FB_AlarmCodeManager(
bAlarm1         :=MesIO_SUBMV_EL1809_1[ 1].value , // SUBMV.-EL1809-ID:1-Input:1 : MV Feeder 1 Opened #Interface
bAlarm2         :=MesIO_SUBMV_EL1809_1[ 2].value , //SUBMV.-EL1809-ID:1-Input:2 : MV Feeder 2 Opened #Interface
bAlarm3         :=MesIO_SUBMV_EL1809_1[ 3].value , //SUBMV.-EL1809-ID:1-Input:3 : MV Feeder 3 Opened  #Interface
bAlarm4         :=MesIO_SUBMV_EL1809_1[ 4].value , //SUBMV.-EL1809-ID:1-Input:4 : Main MVCB Opened #Interface
bAlarm5         :=MesIO_SUBMV_EL1809_1[ 5].value , //SUBMV.-EL1809-ID:1-Input:5 : MainMVCB Tripped #Interface
bAlarm6         :=MesIO_SUBMV_EL1809_1[ 6].value , //SUBMV.-EL1809-ID:1-Input:6 : MainMVCB Earthing #Interface
bAlarm7         :=MesIO_SUBMV_EL1809_1[ 7].value , //SUBMV.-EL1809-ID:1-Input:7 : MainMVCB selector in local position #Interface
bAlarm8         :=MesIO_SUBMV_EL1809_1[ 8].value , //SUBMV.-EL1809-ID:1-Input:8 : MainMVCB motorization in fault #Interface
bAlarm9         :=MesIO_SUBMV_EL1809_1[ 9].value , //SUBMV.-EL1809-ID:1-Input:9 : MV Feeder 1 Tripped #Interface
bAlarm10         :=MesIO_SUBMV_EL1809_1[ 10].value , //SUBMV.-EL1809-ID:1-Input:10 : MV Feeder 2 Tripped #Interface
bAlarm11         :=MesIO_SUBMV_EL1809_1[ 11].value , //SUBMV.-EL1809-ID:1-Input:11 : MV Feeder 3 Tripped  #Interface
bAlarm12         :=MesIO_SUBMV_EL1809_1[ 12].value , //SUBMV.-EL1809-ID:1-Input:12 : MV Feeder 1 Motorization fault #Interface
bAlarm13         :=MesIO_SUBMV_EL1809_1[ 13].value , //SUBMV.-EL1809-ID:1-Input:13 : MV Feeder 2 Motorization fault #Interface
bAlarm14         :=MesIO_SUBMV_EL1809_1[ 14].value , //SUBMV.-EL1809-ID:1-Input:14 : MV Feeder 3 Motorization fault  #Interface
bAlarm15         :=MesIO_SUBMV_EL1809_1[ 15].value , //SUBMV.-EL1809-ID:1-Input:15 : MV Feeder 1 Earthing #Interface
wAlarmCode      => MesData.MesEventCode[1]);   
FB_AlarmCodeManager(
bAlarm1         :=MesIO_SUBMV_EL1809_1[ 16].value , //SUBMV.-EL1809-ID:1-Input:16 : MV Feeder 2 Earthing #Interface
bAlarm2         :=MesIO_SUBMV_EL1809_2[ 1].value , //SUBMV.-EL1809-ID:2-Input:1 : MV Feeder 3 Earthing  #Interface
bAlarm3         :=MesIO_SUBMV_EL1809_2[ 2].value , //SUBMV.-EL1809-ID:2-Input:2 : MV Feeder 1 Selector in local position #Interface
bAlarm4         :=MesIO_SUBMV_EL1809_2[ 3].value , //SUBMV.-EL1809-ID:2-Input:3 : MV Feeder 2 Selector in local position #Interface
bAlarm5         :=MesIO_SUBMV_EL1809_2[ 4].value , //SUBMV.-EL1809-ID:2-Input:4 : MV Feeder 3 Selector in local position  #Interface
bAlarm6         :=MesIO_SUBMV_EL1809_2[ 5].value , //SUBMV.-EL1809-ID:2-Input:5 : Grid MV CB opened #Interface
bAlarm7         :=MesIO_SUBMV_EL1809_2[ 6].value , //SUBMV.-EL1809-ID:2-Input:6 : Measure MV CB opened  #Interface
bAlarm8         :=MesIO_SUBMV_EL1809_2[ 7].value , //SUBMV.-EL1809-ID:2-Input:7 : Measure MV CB Fuse is burned #Interface
bAlarm9         :=MesIO_SUBMV_EL1809_2[ 8].value , //SUBMV.-EL1809-ID:2-Input:8 : Measure MVCB Earthing #Interface
bAlarm10         :=MesIO_SUBMV_EL1809_2[ 9].value , //SUBMV.-EL1809-ID:2-Input:9 : AuxMVCB opened #Interface
bAlarm11         :=MesIO_SUBMV_EL1809_2[ 10].value , //SUBMV.-EL1809-ID:2-Input:10 : AuxMVCB fuse is burned #Interface
bAlarm12         :=MesIO_SUBMV_EL1809_2[ 11].value , //SUBMV.-EL1809-ID:2-Input:11 : AuxMVCB earthing #Interface
bAlarm13         :=MesIO_SUBMV_EL1809_2[ 12].value , //SUBMV.-EL1809-ID:2-Input:12 : Emergency Stop in LV Area #Interface
bAlarm14         :=MesIO_SUBMV_EL1809_2[ 13].value , //SUBMV.-EL1809-ID:2-Input:13 : Emergency stop in MV Area #Interface
bAlarm15         :=MesIO_SUBMV_EL1809_2[ 14].value , //SUBMV.-EL1809-ID:2-Input:14 : Smoke detector in LV Area #Interface
wAlarmCode      => MesData.MesEventCode[2]);   
FB_AlarmCodeManager(
bAlarm1         :=MesIO_SUBMV_EL1809_2[ 16].value , //SUBMV.-EL1809-ID:2-Input:16 : Transformer Alarm synthesis #Interface
bAlarm2         :=MesIO_SUBMV_EL1809_3[ 1].value , //SUBMV.-EL1809-ID:3-Input:1 : Transformer pressure alarm #Interface
bAlarm3         :=MesIO_SUBMV_EL1809_3[ 2].value , //SUBMV.-EL1809-ID:3-Input:2 : Transformer gaz alarm  #Interface
bAlarm4         :=MesIO_SUBMV_EL1809_3[ 3].value , //SUBMV.-EL1809-ID:3-Input:3 : Transformer temperature warning  #Interface
bAlarm5         :=MesIO_SUBMV_EL1809_3[ 4].value , //SUBMV.-EL1809-ID:3-Input:4 : Transformer temperature alarm #Interface
bAlarm6         :=MesIO_SUBMV_EL1809_3[ 5].value , //SUBMV.-EL1809-ID:3-Input:5 : UPS Decharge Batterie State #Interface
bAlarm7         :=MesIO_SUBMV_EL1809_3[ 6].value , //SUBMV.-EL1809-ID:3-Input:6 : UPS alarm synthesis #Interface
bAlarm8         :=MesIO_SUBMV_EL1809_3[ 7].value , //SUBMV.-EL1809-ID:3-Input:7 : UPS  Low Voltage  #Interface
bAlarm9         :=MesIO_SUBMV_EL1809_3[ 8].value , //SUBMV.-EL1809-ID:3-Input:8 : ProtectRelay I>>0 Fault #Interface
bAlarm10         :=MesIO_SUBMV_EL1809_3[ 9].value , //SUBMV.-EL1809-ID:3-Input:9 : ProtectRelay Min U Fault #Interface
bAlarm11         :=MesIO_SUBMV_EL2809_4[ 1].value , //SUBMV.-EL2809-ID:4-Output:1 : MainMVCB Open order #Interface
bAlarm12         :=MesIO_SUBMV_EL2809_4[ 2].value , //SUBMV.-EL2809-ID:4-Output:2 : MainMVCB Close order #Interface
bAlarm13         :=MesIO_SUBMV_EL2809_4[ 3].value , //SUBMV.-EL2809-ID:4-Output:3 : MV Feeder 1 Close Command #Interface
bAlarm14         :=MesIO_SUBMV_EL2809_4[ 4].value , //SUBMV.-EL2809-ID:4-Output:4 : MV Feeder 2 Close Command #Interface
bAlarm15         :=MesIO_SUBMV_EL2809_4[ 5].value , //SUBMV.-EL2809-ID:4-Output:5 : MV Feeder 3 Close Command  #Interface
wAlarmCode      => MesData.MesEventCode[3]);   
FB_AlarmCodeManager(
bAlarm1         :=MesIO_SUBMV_EL2809_4[ 6].value , //SUBMV.-EL2809-ID:4-Output:6 : MV Feeder 1 Open Command #Interface
bAlarm2         :=MesIO_SUBMV_EL2809_4[ 7].value , //SUBMV.-EL2809-ID:4-Output:7 : MV Feeder 2 Open Command #Interface
bAlarm3         :=MesIO_SUBMV_EL2809_4[ 8].value , //SUBMV.-EL2809-ID:4-Output:8 : MV Feeder 3 Open Command  #Interface
bAlarm4         :=MesIO_PTR_1_EL1809_9[ 1].value , //PTR.1-EL1809-ID:9-Input:1 : Motorization alarm MainMVCB #Interface
bAlarm5         :=MesIO_PTR_1_EL1809_9[ 2].value , //PTR.1-EL1809-ID:9-Input:2 : Main MVCB Tripped #Interface
bAlarm6         :=MesIO_PTR_1_EL1809_9[ 3].value , //PTR.1-EL1809-ID:9-Input:3 : MainMVCB selector in Local position #Interface
bAlarm7         :=MesIO_PTR_1_EL1809_9[ 4].value , //PTR.1-EL1809-ID:9-Input:4 : MainMVCB connected to the Earth #Interface
bAlarm8         :=MesIO_PTR_1_EL1809_9[ 5].value , //PTR.1-EL1809-ID:9-Input:5 : Transfo smoke detector 1 #Interface
bAlarm9         :=MesIO_PTR_1_EL1809_9[ 6].value , //PTR.1-EL1809-ID:9-Input:6 : Inverter smoke detector 2 #Interface
bAlarm10         :=MesIO_PTR_1_EL1809_9[ 7].value , //PTR.1-EL1809-ID:9-Input:7 : Door sensor Transformer  area #Interface
bAlarm11         :=MesIO_PTR_1_EL1809_9[ 8].value , //PTR.1-EL1809-ID:9-Input:8 : Door sensor inverter area #Interface
bAlarm12         :=MesIO_PTR_1_EL1809_9[ 9].value , //PTR.1-EL1809-ID:9-Input:9 : Transformer Alarm synthesis #Interface
bAlarm13         :=MesIO_PTR_1_EL1809_9[ 10].value , //PTR.1-EL1809-ID:9-Input:10 : Transformer pressure alarm #Interface
bAlarm14         :=MesIO_PTR_1_EL1809_9[ 11].value , //PTR.1-EL1809-ID:9-Input:11 : Transformer gaz alarm  #Interface
bAlarm15         :=MesIO_PTR_1_EL1809_9[ 12].value , //PTR.1-EL1809-ID:9-Input:12 : Transformer temperature warning  #Interface
wAlarmCode      => MesData.MesEventCode[4]);   
FB_AlarmCodeManager(
bAlarm1         :=MesIO_PTR_1_EL1809_9[ 13].value , //PTR.1-EL1809-ID:9-Input:13 : Transformer temperature alarm #Interface
bAlarm2         :=MesIO_PTR_1_EL1809_9[ 14].value , //PTR.1-EL1809-ID:9-Input:14 : Auxiliairy main CB Opened #Interface
bAlarm3         :=MesIO_PTR_1_EL2809_10[ 1].value , //PTR.1-EL2809-ID:10-Output:1 : Open Command MainMVCB #Interface
bAlarm4         :=MesIO_PTR_1_EL2809_10[ 2].value , //PTR.1-EL2809-ID:10-Output:2 : Close Command MainMVCB #Interface
bAlarm5         :=MesIO_PTR_2_EL1809_9[ 1].value , //PTR.2-EL1809-ID:9-Input:1 : Motorization alarm MainMVCB #Interface
bAlarm6         :=MesIO_PTR_2_EL1809_9[ 2].value , //PTR.2-EL1809-ID:9-Input:2 : Main MVCB Tripped #Interface
bAlarm7         :=MesIO_PTR_2_EL1809_9[ 3].value , //PTR.2-EL1809-ID:9-Input:3 : MainMVCB selector in Local position #Interface
bAlarm8         :=MesIO_PTR_2_EL1809_9[ 4].value , //PTR.2-EL1809-ID:9-Input:4 : MainMVCB connected to the Earth #Interface
bAlarm9         :=MesIO_PTR_2_EL1809_9[ 5].value , //PTR.2-EL1809-ID:9-Input:5 : Transfo smoke detector 1 #Interface
bAlarm10         :=MesIO_PTR_2_EL1809_9[ 6].value , //PTR.2-EL1809-ID:9-Input:6 : Inverter smoke detector 2 #Interface
bAlarm11         :=MesIO_PTR_2_EL1809_9[ 7].value , //PTR.2-EL1809-ID:9-Input:7 : Door sensor Transformer  area #Interface
bAlarm12         :=MesIO_PTR_2_EL1809_9[ 8].value , //PTR.2-EL1809-ID:9-Input:8 : Door sensor inverter area #Interface
bAlarm13         :=MesIO_PTR_2_EL1809_9[ 9].value , //PTR.2-EL1809-ID:9-Input:9 : Transformer Alarm synthesis #Interface
bAlarm14         :=MesIO_PTR_2_EL1809_9[ 10].value , //PTR.2-EL1809-ID:9-Input:10 : Transformer pressure alarm #Interface
bAlarm15         :=MesIO_PTR_2_EL1809_9[ 11].value , //PTR.2-EL1809-ID:9-Input:11 : Transformer gaz alarm  #Interface
wAlarmCode      => MesData.MesEventCode[5]);   
FB_AlarmCodeManager(
bAlarm1         :=MesIO_PTR_2_EL1809_9[ 12].value , //PTR.2-EL1809-ID:9-Input:12 : Transformer temperature warning  #Interface
bAlarm2         :=MesIO_PTR_2_EL1809_9[ 13].value , //PTR.2-EL1809-ID:9-Input:13 : Transformer temperature alarm #Interface
bAlarm3         :=MesIO_PTR_2_EL1809_9[ 14].value , //PTR.2-EL1809-ID:9-Input:14 : Auxiliairy main CB Opened #Interface
bAlarm4         :=MesIO_PTR_2_EL2809_10[ 1].value , //PTR.2-EL2809-ID:10-Output:1 : Open Command MainMVCB #Interface
bAlarm5         :=MesIO_PTR_2_EL2809_10[ 2].value , //PTR.2-EL2809-ID:10-Output:2 : Close Command MainMVCB #Interface
bAlarm6         :=MesIO_PTR_3_EL1809_9[ 1].value , //PTR.3-EL1809-ID:9-Input:1 : Motorization alarm MainMVCB #Interface
bAlarm7         :=MesIO_PTR_3_EL1809_9[ 2].value , //PTR.3-EL1809-ID:9-Input:2 : Main MVCB Tripped #Interface
bAlarm8         :=MesIO_PTR_3_EL1809_9[ 3].value , //PTR.3-EL1809-ID:9-Input:3 : MainMVCB selector in Local position #Interface
bAlarm9         :=MesIO_PTR_3_EL1809_9[ 4].value , //PTR.3-EL1809-ID:9-Input:4 : MainMVCB connected to the Earth #Interface
bAlarm10         :=MesIO_PTR_3_EL1809_9[ 5].value , //PTR.3-EL1809-ID:9-Input:5 : Transfo smoke detector 1 #Interface
bAlarm11         :=MesIO_PTR_3_EL1809_9[ 6].value , //PTR.3-EL1809-ID:9-Input:6 : Inverter smoke detector 2 #Interface
bAlarm12         :=MesIO_PTR_3_EL1809_9[ 7].value , //PTR.3-EL1809-ID:9-Input:7 : Door sensor Transformer  area #Interface
bAlarm13         :=MesIO_PTR_3_EL1809_9[ 8].value , //PTR.3-EL1809-ID:9-Input:8 : Door sensor inverter area #Interface
bAlarm14         :=MesIO_PTR_3_EL1809_9[ 9].value , //PTR.3-EL1809-ID:9-Input:9 : Transformer Alarm synthesis #Interface
bAlarm15         :=MesIO_PTR_3_EL1809_9[ 10].value , //PTR.3-EL1809-ID:9-Input:10 : Transformer pressure alarm #Interface
wAlarmCode      => MesData.MesEventCode[6]);   
FB_AlarmCodeManager(
bAlarm1         :=MesIO_PTR_3_EL1809_9[ 11].value , //PTR.3-EL1809-ID:9-Input:11 : Transformer gaz alarm  #Interface
bAlarm2         :=MesIO_PTR_3_EL1809_9[ 12].value , //PTR.3-EL1809-ID:9-Input:12 : Transformer temperature warning  #Interface
bAlarm3         :=MesIO_PTR_3_EL1809_9[ 13].value , //PTR.3-EL1809-ID:9-Input:13 : Transformer temperature alarm #Interface
bAlarm4         :=MesIO_PTR_3_EL1809_9[ 14].value , //PTR.3-EL1809-ID:9-Input:14 : Auxiliairy main CB Opened #Interface
bAlarm5         :=MesIO_PTR_3_EL2809_10[ 1].value , //PTR.3-EL2809-ID:10-Output:1 : Open Command MainMVCB #Interface
bAlarm6         :=MesIO_PTR_3_EL2809_10[ 2].value , //PTR.3-EL2809-ID:10-Output:2 : Close Command MainMVCB #Interface
wAlarmCode      => MesData.MesEventCode[7]);
END_METHOD

METHOD M_Evaluate : BOOL
(*
MesIO_SUBMV_EL1809_1[1].value := axDI[1] ;
MesIO_SUBMV_EL1809_1[2].value := axDI[2] ;
MesIO_SUBMV_EL1809_1[3].value := axDI[3] ;
MesIO_SUBMV_EL1809_1[4].value := axDI[4] ;
MesIO_SUBMV_EL1809_1[5].value := axDI[5] ;
MesIO_SUBMV_EL1809_1[6].value := axDI[6] ;
MesIO_SUBMV_EL1809_1[7].value := axDI[7] ;
MesIO_SUBMV_EL1809_1[8].value := axDI[8] ;
MesIO_SUBMV_EL1809_1[9].value := axDI[9] ;
MesIO_SUBMV_EL1809_1[10].value := axDI[10] ;
MesIO_SUBMV_EL1809_1[11].value := axDI[11] ;
MesIO_SUBMV_EL1809_1[12].value := axDI[12] ;
MesIO_SUBMV_EL1809_1[13].value := axDI[13] ;
MesIO_SUBMV_EL1809_1[14].value := axDI[14] ;
MesIO_SUBMV_EL1809_1[15].value := axDI[15] ;
MesIO_SUBMV_EL1809_1[16].value := axDI[16] ;
MesIO_SUBMV_EL1809_2[1].value := axDI[17] ;
MesIO_SUBMV_EL1809_2[2].value := axDI[18] ;
MesIO_SUBMV_EL1809_2[3].value := axDI[19] ;
MesIO_SUBMV_EL1809_2[4].value := axDI[20] ;
MesIO_SUBMV_EL1809_2[5].value := axDI[21] ;
MesIO_SUBMV_EL1809_2[6].value := axDI[22] ;
MesIO_SUBMV_EL1809_2[7].value := axDI[23] ;
MesIO_SUBMV_EL1809_2[8].value := axDI[24] ;
MesIO_SUBMV_EL1809_2[9].value := axDI[25] ;
MesIO_SUBMV_EL1809_2[10].value := axDI[26] ;
MesIO_SUBMV_EL1809_2[11].value := axDI[27] ;
MesIO_SUBMV_EL1809_2[12].value := axDI[28] ;
MesIO_SUBMV_EL1809_2[13].value := axDI[29] ;
MesIO_SUBMV_EL1809_2[14].value := axDI[30] ;
MesIO_SUBMV_EL1809_2[15].value := axDI[31] ;
MesIO_SUBMV_EL1809_2[16].value := axDI[32] ;
MesIO_SUBMV_EL1809_3[1].value := axDI[33] ;
MesIO_SUBMV_EL1809_3[2].value := axDI[34] ;
MesIO_SUBMV_EL1809_3[3].value := axDI[35] ;
MesIO_SUBMV_EL1809_3[4].value := axDI[36] ;
MesIO_SUBMV_EL1809_3[5].value := axDI[37] ;
MesIO_SUBMV_EL1809_3[6].value := axDI[38] ;
MesIO_SUBMV_EL1809_3[7].value := axDI[39] ;
MesIO_SUBMV_EL1809_3[8].value := axDI[40] ;
MesIO_SUBMV_EL1809_3[9].value := axDI[41] ;
MesIO_SUBMV_EL1809_3[10].value := axDI[42] ;
MesIO_SUBMV_EL1809_3[11].value := axDI[43] ;
MesIO_SUBMV_EL1809_3[12].value := axDI[44] ;
MesIO_SUBMV_EL1809_3[13].value := axDI[45] ;
MesIO_SUBMV_EL1809_3[14].value := axDI[46] ;
MesIO_SUBMV_EL1809_3[15].value := axDI[47] ;
MesIO_SUBMV_EL1809_3[16].value := axDI[48] ;
axDO[1] := MesIO_SUBMV_EL2809_4[1].value ; 
axDO[2] := MesIO_SUBMV_EL2809_4[2].value ; 
axDO[3] := MesIO_SUBMV_EL2809_4[3].value ; 
axDO[4] := MesIO_SUBMV_EL2809_4[4].value ; 
axDO[5] := MesIO_SUBMV_EL2809_4[5].value ; 
axDO[6] := MesIO_SUBMV_EL2809_4[6].value ; 
axDO[7] := MesIO_SUBMV_EL2809_4[7].value ; 
axDO[8] := MesIO_SUBMV_EL2809_4[8].value ; 
axDO[9] := MesIO_SUBMV_EL2809_4[9].value ; 
axDO[10] := MesIO_SUBMV_EL2809_4[10].value ; 
axDO[11] := MesIO_SUBMV_EL2809_4[11].value ; 
axDO[12] := MesIO_SUBMV_EL2809_4[12].value ; 
axDO[13] := MesIO_SUBMV_EL2809_4[13].value ; 
axDO[14] := MesIO_SUBMV_EL2809_4[14].value ; 
axDO[15] := MesIO_SUBMV_EL2809_4[15].value ; 
axDO[16] := MesIO_SUBMV_EL2809_4[16].value ; 
MesIO_SUBMV_EL3024_5[1].value := axAI[1] ;
MesIO_SUBMV_EL3024_5[2].value := axAI[2] ;
MesIO_SUBMV_EL3024_5[3].value := axAI[3] ;
MesIO_SUBMV_EL3024_5[4].value := axAI[4] ;
MesIO_PTR_1_EL3024_8[1].value := axAI[5] ;
MesIO_PTR_1_EL3024_8[2].value := axAI[6] ;
MesIO_PTR_1_EL3024_8[3].value := axAI[7] ;
MesIO_PTR_1_EL3024_8[4].value := axAI[8] ;
MesIO_PTR_1_EL1809_9[1].value := axDI[49] ;
MesIO_PTR_1_EL1809_9[2].value := axDI[50] ;
MesIO_PTR_1_EL1809_9[3].value := axDI[51] ;
MesIO_PTR_1_EL1809_9[4].value := axDI[52] ;
MesIO_PTR_1_EL1809_9[5].value := axDI[53] ;
MesIO_PTR_1_EL1809_9[6].value := axDI[54] ;
MesIO_PTR_1_EL1809_9[7].value := axDI[55] ;
MesIO_PTR_1_EL1809_9[8].value := axDI[56] ;
MesIO_PTR_1_EL1809_9[9].value := axDI[57] ;
MesIO_PTR_1_EL1809_9[10].value := axDI[58] ;
MesIO_PTR_1_EL1809_9[11].value := axDI[59] ;
MesIO_PTR_1_EL1809_9[12].value := axDI[60] ;
MesIO_PTR_1_EL1809_9[13].value := axDI[61] ;
MesIO_PTR_1_EL1809_9[14].value := axDI[62] ;
MesIO_PTR_1_EL1809_9[15].value := axDI[63] ;
MesIO_PTR_1_EL1809_9[16].value := axDI[64] ;
axDO[17] := MesIO_PTR_1_EL2809_10[1].value ; 
axDO[18] := MesIO_PTR_1_EL2809_10[2].value ; 
axDO[19] := MesIO_PTR_1_EL2809_10[3].value ; 
axDO[20] := MesIO_PTR_1_EL2809_10[4].value ; 
axDO[21] := MesIO_PTR_1_EL2809_10[5].value ; 
axDO[22] := MesIO_PTR_1_EL2809_10[6].value ; 
axDO[23] := MesIO_PTR_1_EL2809_10[7].value ; 
axDO[24] := MesIO_PTR_1_EL2809_10[8].value ; 
axDO[25] := MesIO_PTR_1_EL2809_10[9].value ; 
axDO[26] := MesIO_PTR_1_EL2809_10[10].value ; 
axDO[27] := MesIO_PTR_1_EL2809_10[11].value ; 
axDO[28] := MesIO_PTR_1_EL2809_10[12].value ; 
axDO[29] := MesIO_PTR_1_EL2809_10[13].value ; 
axDO[30] := MesIO_PTR_1_EL2809_10[14].value ; 
axDO[31] := MesIO_PTR_1_EL2809_10[15].value ; 
axDO[32] := MesIO_PTR_1_EL2809_10[16].value ; 
MesIO_PTR_2_EL3024_8[1].value := axAI[9] ;
MesIO_PTR_2_EL3024_8[2].value := axAI[10] ;
MesIO_PTR_2_EL3024_8[3].value := axAI[11] ;
MesIO_PTR_2_EL3024_8[4].value := axAI[12] ;
MesIO_PTR_2_EL1809_9[1].value := axDI[65] ;
MesIO_PTR_2_EL1809_9[2].value := axDI[66] ;
MesIO_PTR_2_EL1809_9[3].value := axDI[67] ;
MesIO_PTR_2_EL1809_9[4].value := axDI[68] ;
MesIO_PTR_2_EL1809_9[5].value := axDI[69] ;
MesIO_PTR_2_EL1809_9[6].value := axDI[70] ;
MesIO_PTR_2_EL1809_9[7].value := axDI[71] ;
MesIO_PTR_2_EL1809_9[8].value := axDI[72] ;
MesIO_PTR_2_EL1809_9[9].value := axDI[73] ;
MesIO_PTR_2_EL1809_9[10].value := axDI[74] ;
MesIO_PTR_2_EL1809_9[11].value := axDI[75] ;
MesIO_PTR_2_EL1809_9[12].value := axDI[76] ;
MesIO_PTR_2_EL1809_9[13].value := axDI[77] ;
MesIO_PTR_2_EL1809_9[14].value := axDI[78] ;
MesIO_PTR_2_EL1809_9[15].value := axDI[79] ;
MesIO_PTR_2_EL1809_9[16].value := axDI[80] ;
axDO[33] := MesIO_PTR_2_EL2809_10[1].value ; 
axDO[34] := MesIO_PTR_2_EL2809_10[2].value ; 
axDO[35] := MesIO_PTR_2_EL2809_10[3].value ; 
axDO[36] := MesIO_PTR_2_EL2809_10[4].value ; 
axDO[37] := MesIO_PTR_2_EL2809_10[5].value ; 
axDO[38] := MesIO_PTR_2_EL2809_10[6].value ; 
axDO[39] := MesIO_PTR_2_EL2809_10[7].value ; 
axDO[40] := MesIO_PTR_2_EL2809_10[8].value ; 
axDO[41] := MesIO_PTR_2_EL2809_10[9].value ; 
axDO[42] := MesIO_PTR_2_EL2809_10[10].value ; 
axDO[43] := MesIO_PTR_2_EL2809_10[11].value ; 
axDO[44] := MesIO_PTR_2_EL2809_10[12].value ; 
axDO[45] := MesIO_PTR_2_EL2809_10[13].value ; 
axDO[46] := MesIO_PTR_2_EL2809_10[14].value ; 
axDO[47] := MesIO_PTR_2_EL2809_10[15].value ; 
axDO[48] := MesIO_PTR_2_EL2809_10[16].value ; 
MesIO_PTR_3_EL3024_8[1].value := axAI[13] ;
MesIO_PTR_3_EL3024_8[2].value := axAI[14] ;
MesIO_PTR_3_EL3024_8[3].value := axAI[15] ;
MesIO_PTR_3_EL3024_8[4].value := axAI[16] ;
MesIO_PTR_3_EL1809_9[1].value := axDI[81] ;
MesIO_PTR_3_EL1809_9[2].value := axDI[82] ;
MesIO_PTR_3_EL1809_9[3].value := axDI[83] ;
MesIO_PTR_3_EL1809_9[4].value := axDI[84] ;
MesIO_PTR_3_EL1809_9[5].value := axDI[85] ;
MesIO_PTR_3_EL1809_9[6].value := axDI[86] ;
MesIO_PTR_3_EL1809_9[7].value := axDI[87] ;
MesIO_PTR_3_EL1809_9[8].value := axDI[88] ;
MesIO_PTR_3_EL1809_9[9].value := axDI[89] ;
MesIO_PTR_3_EL1809_9[10].value := axDI[90] ;
MesIO_PTR_3_EL1809_9[11].value := axDI[91] ;
MesIO_PTR_3_EL1809_9[12].value := axDI[92] ;
MesIO_PTR_3_EL1809_9[13].value := axDI[93] ;
MesIO_PTR_3_EL1809_9[14].value := axDI[94] ;
MesIO_PTR_3_EL1809_9[15].value := axDI[95] ;
MesIO_PTR_3_EL1809_9[16].value := axDI[96] ;
axDO[49] := MesIO_PTR_3_EL2809_10[1].value ; 
axDO[50] := MesIO_PTR_3_EL2809_10[2].value ; 
axDO[51] := MesIO_PTR_3_EL2809_10[3].value ; 
axDO[52] := MesIO_PTR_3_EL2809_10[4].value ; 
axDO[53] := MesIO_PTR_3_EL2809_10[5].value ; 
axDO[54] := MesIO_PTR_3_EL2809_10[6].value ; 
axDO[55] := MesIO_PTR_3_EL2809_10[7].value ; 
axDO[56] := MesIO_PTR_3_EL2809_10[8].value ; 
axDO[57] := MesIO_PTR_3_EL2809_10[9].value ; 
axDO[58] := MesIO_PTR_3_EL2809_10[10].value ; 
axDO[59] := MesIO_PTR_3_EL2809_10[11].value ; 
axDO[60] := MesIO_PTR_3_EL2809_10[12].value ; 
axDO[61] := MesIO_PTR_3_EL2809_10[13].value ; 
axDO[62] := MesIO_PTR_3_EL2809_10[14].value ; 
axDO[63] := MesIO_PTR_3_EL2809_10[15].value ; 
axDO[64] := MesIO_PTR_3_EL2809_10[16].value ; 
*)
END_METHOD

METHOD M_Init : BOOL
VAR
	KK : BYTE;
END_VAR

MesIO_SUBMV_EL1809_1[ 1].Description := 'MV Feeder 1 Opened' ; 
MesIO_SUBMV_EL1809_1[ 2].Description := 'MV Feeder 2 Opened' ; 
MesIO_SUBMV_EL1809_1[ 3].Description := 'MV Feeder 3 Opened ' ; 
MesIO_SUBMV_EL1809_1[ 4].Description := 'Main MVCB Opened' ; 
MesIO_SUBMV_EL1809_1[ 5].Description := 'MainMVCB Tripped' ; 
MesIO_SUBMV_EL1809_1[ 6].Description := 'MainMVCB Earthing' ; 
MesIO_SUBMV_EL1809_1[ 7].Description := 'MainMVCB selector in local position' ; 
MesIO_SUBMV_EL1809_1[ 8].Description := 'MainMVCB motorization in fault' ; 
MesIO_SUBMV_EL1809_1[ 9].Description := 'MV Feeder 1 Tripped' ; 
MesIO_SUBMV_EL1809_1[ 10].Description := 'MV Feeder 2 Tripped' ; 
MesIO_SUBMV_EL1809_1[ 11].Description := 'MV Feeder 3 Tripped ' ; 
MesIO_SUBMV_EL1809_1[ 12].Description := 'MV Feeder 1 Motorization fault' ; 
MesIO_SUBMV_EL1809_1[ 13].Description := 'MV Feeder 2 Motorization fault' ; 
MesIO_SUBMV_EL1809_1[ 14].Description := 'MV Feeder 3 Motorization fault ' ; 
MesIO_SUBMV_EL1809_1[ 15].Description := 'MV Feeder 1 Earthing' ; 
MesIO_SUBMV_EL1809_1[ 16].Description := 'MV Feeder 2 Earthing' ; 
MesIO_SUBMV_EL1809_2[ 1].Description := 'MV Feeder 3 Earthing ' ; 
MesIO_SUBMV_EL1809_2[ 2].Description := 'MV Feeder 1 Selector in local position' ; 
MesIO_SUBMV_EL1809_2[ 3].Description := 'MV Feeder 2 Selector in local position' ; 
MesIO_SUBMV_EL1809_2[ 4].Description := 'MV Feeder 3 Selector in local position ' ; 
MesIO_SUBMV_EL1809_2[ 5].Description := 'Grid MV CB opened' ; 
MesIO_SUBMV_EL1809_2[ 6].Description := 'Measure MV CB opened ' ; 
MesIO_SUBMV_EL1809_2[ 7].Description := 'Measure MV CB Fuse is burned' ; 
MesIO_SUBMV_EL1809_2[ 8].Description := 'Measure MVCB Earthing' ; 
MesIO_SUBMV_EL1809_2[ 9].Description := 'AuxMVCB opened' ; 
MesIO_SUBMV_EL1809_2[ 10].Description := 'AuxMVCB fuse is burned' ; 
MesIO_SUBMV_EL1809_2[ 11].Description := 'AuxMVCB earthing' ; 
MesIO_SUBMV_EL1809_2[ 12].Description := 'Emergency Stop in LV Area' ; 
MesIO_SUBMV_EL1809_2[ 13].Description := 'Emergency stop in MV Area' ; 
MesIO_SUBMV_EL1809_2[ 14].Description := 'Smoke detector in LV Area' ; 
MesIO_SUBMV_EL1809_2[ 16].Description := 'Transformer Alarm synthesis' ; 
MesIO_SUBMV_EL1809_3[ 1].Description := 'Transformer pressure alarm' ; 
MesIO_SUBMV_EL1809_3[ 2].Description := 'Transformer gaz alarm ' ; 
MesIO_SUBMV_EL1809_3[ 3].Description := 'Transformer temperature warning ' ; 
MesIO_SUBMV_EL1809_3[ 4].Description := 'Transformer temperature alarm' ; 
MesIO_SUBMV_EL1809_3[ 5].Description := 'UPS Decharge Batterie State' ; 
MesIO_SUBMV_EL1809_3[ 6].Description := 'UPS alarm synthesis' ; 
MesIO_SUBMV_EL1809_3[ 7].Description := 'UPS  Low Voltage ' ; 
MesIO_SUBMV_EL1809_3[ 8].Description := 'ProtectRelay I>>0 Fault' ; 
MesIO_SUBMV_EL1809_3[ 9].Description := 'ProtectRelay Min U Fault' ; 
MesIO_SUBMV_EL2809_4[ 1].Description := 'MainMVCB Open order' ; 
MesIO_SUBMV_EL2809_4[ 2].Description := 'MainMVCB Close order' ; 
MesIO_SUBMV_EL2809_4[ 3].Description := 'MV Feeder 1 Close Command' ; 
MesIO_SUBMV_EL2809_4[ 4].Description := 'MV Feeder 2 Close Command' ; 
MesIO_SUBMV_EL2809_4[ 5].Description := 'MV Feeder 3 Close Command ' ; 
MesIO_SUBMV_EL2809_4[ 6].Description := 'MV Feeder 1 Open Command' ; 
MesIO_SUBMV_EL2809_4[ 7].Description := 'MV Feeder 2 Open Command' ; 
MesIO_SUBMV_EL2809_4[ 8].Description := 'MV Feeder 3 Open Command ' ; 
MesIO_SUBMV_EL3024_5[ 1].Description := 'Pyranometer GHI' ; 
MesIO_SUBMV_EL3024_5[ 2].Description := 'Pyranometer GTI' ; 
MesIO_SUBMV_EL3024_5[ 3].Description := 'External Temperature' ; 
MesIO_SUBMV_EL3024_5[ 4].Description := 'External Hygrometry' ; 
MesIO_SUBMV_EL3024_5[ 1].Description := 'Wind direction ' ; 
MesIO_SUBMV_EL3024_5[ 2].Description := 'Wind Speed' ; 
MesIO_PTR_1_EL3024_8[ 1].Description := 'Panel Temperature sensor 1' ; 
MesIO_PTR_1_EL3024_8[ 2].Description := 'Panel Temperature sensor 2' ; 
MesIO_PTR_1_EL3024_8[ 3].Description := 'Pyranometer GTI' ; 
MesIO_PTR_1_EL1809_9[ 1].Description := 'Motorization alarm MainMVCB' ; 
MesIO_PTR_1_EL1809_9[ 2].Description := 'Main MVCB Tripped' ; 
MesIO_PTR_1_EL1809_9[ 3].Description := 'MainMVCB selector in Local position' ; 
MesIO_PTR_1_EL1809_9[ 4].Description := 'MainMVCB connected to the Earth' ; 
MesIO_PTR_1_EL1809_9[ 5].Description := 'Transfo smoke detector 1' ; 
MesIO_PTR_1_EL1809_9[ 6].Description := 'Inverter smoke detector 2' ; 
MesIO_PTR_1_EL1809_9[ 7].Description := 'Door sensor Transformer  area' ; 
MesIO_PTR_1_EL1809_9[ 8].Description := 'Door sensor inverter area' ; 
MesIO_PTR_1_EL1809_9[ 9].Description := 'Transformer Alarm synthesis' ; 
MesIO_PTR_1_EL1809_9[ 10].Description := 'Transformer pressure alarm' ; 
MesIO_PTR_1_EL1809_9[ 11].Description := 'Transformer gaz alarm ' ; 
MesIO_PTR_1_EL1809_9[ 12].Description := 'Transformer temperature warning ' ; 
MesIO_PTR_1_EL1809_9[ 13].Description := 'Transformer temperature alarm' ; 
MesIO_PTR_1_EL1809_9[ 14].Description := 'Auxiliairy main CB Opened' ; 
MesIO_PTR_1_EL2809_10[ 1].Description := 'Open Command MainMVCB' ; 
MesIO_PTR_1_EL2809_10[ 2].Description := 'Close Command MainMVCB' ; 
MesIO_PTR_2_EL3024_8[ 1].Description := 'Panel Temperature sensor 1' ; 
MesIO_PTR_2_EL3024_8[ 2].Description := 'Panel Temperature sensor 2' ; 
MesIO_PTR_2_EL3024_8[ 3].Description := 'Pyranometer GTI' ; 
MesIO_PTR_2_EL1809_9[ 1].Description := 'Motorization alarm MainMVCB' ; 
MesIO_PTR_2_EL1809_9[ 2].Description := 'Main MVCB Tripped' ; 
MesIO_PTR_2_EL1809_9[ 3].Description := 'MainMVCB selector in Local position' ; 
MesIO_PTR_2_EL1809_9[ 4].Description := 'MainMVCB connected to the Earth' ; 
MesIO_PTR_2_EL1809_9[ 5].Description := 'Transfo smoke detector 1' ; 
MesIO_PTR_2_EL1809_9[ 6].Description := 'Inverter smoke detector 2' ; 
MesIO_PTR_2_EL1809_9[ 7].Description := 'Door sensor Transformer  area' ; 
MesIO_PTR_2_EL1809_9[ 8].Description := 'Door sensor inverter area' ; 
MesIO_PTR_2_EL1809_9[ 9].Description := 'Transformer Alarm synthesis' ; 
MesIO_PTR_2_EL1809_9[ 10].Description := 'Transformer pressure alarm' ; 
MesIO_PTR_2_EL1809_9[ 11].Description := 'Transformer gaz alarm ' ; 
MesIO_PTR_2_EL1809_9[ 12].Description := 'Transformer temperature warning ' ; 
MesIO_PTR_2_EL1809_9[ 13].Description := 'Transformer temperature alarm' ; 
MesIO_PTR_2_EL1809_9[ 14].Description := 'Auxiliairy main CB Opened' ; 
MesIO_PTR_2_EL2809_10[ 1].Description := 'Open Command MainMVCB' ; 
MesIO_PTR_2_EL2809_10[ 2].Description := 'Close Command MainMVCB' ; 
MesIO_PTR_3_EL3024_8[ 1].Description := 'Panel Temperature sensor 1' ; 
MesIO_PTR_3_EL3024_8[ 2].Description := 'Panel Temperature sensor 2' ; 
MesIO_PTR_3_EL3024_8[ 3].Description := 'Pyranometer GTI' ; 
MesIO_PTR_3_EL1809_9[ 1].Description := 'Motorization alarm MainMVCB' ; 
MesIO_PTR_3_EL1809_9[ 2].Description := 'Main MVCB Tripped' ; 
MesIO_PTR_3_EL1809_9[ 3].Description := 'MainMVCB selector in Local position' ; 
MesIO_PTR_3_EL1809_9[ 4].Description := 'MainMVCB connected to the Earth' ; 
MesIO_PTR_3_EL1809_9[ 5].Description := 'Transfo smoke detector 1' ; 
MesIO_PTR_3_EL1809_9[ 6].Description := 'Inverter smoke detector 2' ; 
MesIO_PTR_3_EL1809_9[ 7].Description := 'Door sensor Transformer  area' ; 
MesIO_PTR_3_EL1809_9[ 8].Description := 'Door sensor inverter area' ; 
MesIO_PTR_3_EL1809_9[ 9].Description := 'Transformer Alarm synthesis' ; 
MesIO_PTR_3_EL1809_9[ 10].Description := 'Transformer pressure alarm' ; 
MesIO_PTR_3_EL1809_9[ 11].Description := 'Transformer gaz alarm ' ; 
MesIO_PTR_3_EL1809_9[ 12].Description := 'Transformer temperature warning ' ; 
MesIO_PTR_3_EL1809_9[ 13].Description := 'Transformer temperature alarm' ; 
MesIO_PTR_3_EL1809_9[ 14].Description := 'Auxiliairy main CB Opened' ; 
MesIO_PTR_3_EL2809_10[ 1].Description := 'Open Command MainMVCB' ; 
MesIO_PTR_3_EL2809_10[ 2].Description := 'Close Command MainMVCB' ;
END_METHOD

METHOD M_Inputs
///////////
// Intput interface between POUs and I/O Cards
//////////////

VAR 
KK							: BYTE ; 					// For LOOP 
MesCouplerStateSUB_MV			: ST_AI ; 
END_VAR
END_METHOD

METHOD M_Outputs : BOOL
///////////
// Intput interface between POUs and I/O Cards
//////////////
VAR
	KK	: BYTE;

	A1_MainMVCB: INT;
END_VAR

MesIO_SUBMV_EL2809_4[ 1].value := A1_SUBMV.A1_MainMVCB.OUT_CmdOpen_IO and not IN_CmdInhibOutput_OPC; 
MesIO_SUBMV_EL2809_4[ 2].value := A1_SUBMV.A1_MainMVCB.OUT_CmdClose_IO and not IN_CmdInhibOutput_OPC; 
MesIO_SUBMV_EL2809_4[ 3].value := A1_SUBMV.AX_FeederMVCB[1].OUT_CmdClose_IO and not IN_CmdInhibOutput_OPC; 
MesIO_SUBMV_EL2809_4[ 4].value := A1_SUBMV.AX_FeederMVCB[2].OUT_CmdClose_IO and not IN_CmdInhibOutput_OPC; 
MesIO_SUBMV_EL2809_4[ 5].value := A1_SUBMV.AX_FeederMVCB[3].OUT_CmdClose_IO and not IN_CmdInhibOutput_OPC; 
MesIO_SUBMV_EL2809_4[ 6].value := A1_SUBMV.AX_FeederMVCB[1].OUT_CmdOpen_IO and not IN_CmdInhibOutput_OPC; 
MesIO_SUBMV_EL2809_4[ 7].value := A1_SUBMV.AX_FeederMVCB[2].OUT_CmdOpen_IO and not IN_CmdInhibOutput_OPC; 
MesIO_SUBMV_EL2809_4[ 8].value := A1_SUBMV.AX_FeederMVCB[3].OUT_CmdOpen_IO and not IN_CmdInhibOutput_OPC; 
MesIO_PTR_1_EL2809_10[ 1].value := AX_PTR[1].A1_MainMVCB_PTR.OUT_CmdOpen_IO and not IN_CmdInhibOutput_OPC; 
MesIO_PTR_1_EL2809_10[ 2].value := AX_PTR[1].A1_MainMVCB_PTR.OUT_CmdClose_IO and not IN_CmdInhibOutput_OPC; 
MesIO_PTR_2_EL2809_10[ 1].value := AX_PTR[2].A1_MainMVCB_PTR.OUT_CmdOpen_IO and not IN_CmdInhibOutput_OPC; 
MesIO_PTR_2_EL2809_10[ 2].value := AX_PTR[2].A1_MainMVCB_PTR.OUT_CmdClose_IO and not IN_CmdInhibOutput_OPC; 
MesIO_PTR_3_EL2809_10[ 1].value := AX_PTR[3].A1_MainMVCB_PTR.OUT_CmdOpen_IO and not IN_CmdInhibOutput_OPC; 
MesIO_PTR_3_EL2809_10[ 2].value := AX_PTR[3].A1_MainMVCB_PTR.OUT_CmdClose_IO and not IN_CmdInhibOutput_OPC;
END_METHOD

END_PROGRAM

// ---- 04_Application/HMI/HMI.TcPOU
PROGRAM HMI
VAR_INPUT
	BMS_Display				: BAT_NARADA;
	PCS_Display				: PCS_Sma;
	ESS_Display 			: ESS_Exd;
	
	PTR_Display				: PTR_Exd;
	INV_Display				: INV_Huawei;
	
END_VAR

// HPP
	HPP_HMI();
	
	BESS_HMI();
	
	SPP_HMI();

METHOD M_UserManagement : BOOL
VAR_INPUT
END_VAR
END_METHOD

END_PROGRAM

// ---- 04_Application/HMI/HPP/HPP_HMI.TcPOU
PROGRAM HPP_HMI
VAR
	
	bTrig_SetptP					: BOOL;
	bTrig_SetptQ					: BOOL;
	bTrig_TargetSoCSoC				: BOOL;
	bTrig_TargetSoCP				: BOOL;
	bTrig_FreqRegParam				: BOOL;
	bTrig_UregParam					: BOOL;

	
	SetptP_IO						: REAL;
	SetptQ_IO						: REAL;
	                            	
	CalHppData						: PP;
	KK 								: UINT;
END_VAR

END_PROGRAM

// ---- 04_Application/HMI/BESS/BESS_HMI.TcPOU
PROGRAM BESS_HMI
VAR

	MesP_PowerColPair : REAL;
	MesQ_PowerColPair : REAL;


	StateInv		: STRING;
	PCS_StateInv	: ARRAY[0..100] OF STRING;
	
	
	Pcs_Bat1_On : BOOL;
	Pcs_Bat2_On : BOOL;
	NumBmsDisplayed	: UINT := 1;
	NumPcsDisplayed	: UINT := 1;	
	NumEssDisplayed	: UINT := 1;
		
	BarDisplay_Max	: REAL;
	BarDisplay_Min	: REAL;
	BarDisplay_ID	: UINT := 1; // 1:SoC, 2:Idc, 3: Udc, 4:SoH
	BarDisplay_1	: BOOL := TRUE;
	BarDisplay_2	: BOOL;
	BarDisplay_3	: BOOL;
	BarDisplay_4	: BOOL;
	
	IN_NumSystemSelected		: UINT := 1; // Input : numéro du System sélectionné (sur le nombre total de systèmes)
	ID_ESS_Displayed			: UINT;
	ID_PCS_ESS_Displayed		: UINT; // Identifiant du premier PCS du système
	ID_BAT_ESS_Displayed		: UINT; // Identifiant du premier système BMS du système
	ID_PowerCol_PCS_Displayed	: UINT;	// Identifiant de la première colonne de puissance du système
	
	ParamNbSystemESS : UINT := 1;
	
	// PCS1
		Trig_Pcs1GridFormer		: R_TRIG;
		Trig_Pcs1GridFeeder		: R_TRIG;
		Trig_Pcs1StartOn		: R_TRIG;
		Trig_Pcs1StartOff		: R_TRIG;
		Trig_Pcs1StopOn			: R_TRIG;
		Trig_Pcs1StopOff		: R_TRIG;
		Trig_Pcs1StandbyOn		: R_TRIG;
		Trig_Pcs1StandbyOff		: R_TRIG;
		
		Trig_Pcs1CmdPOn			: R_TRIG;
		Trig_Pcs1CmdPOff		: R_TRIG;
		Trig_Pcs1CmdQOn			: R_TRIG;
		Trig_Pcs1CmdQOff		: R_TRIG;	
		
		Trig_Pcs1CmdLocalOn		: R_TRIG;
		Trig_Pcs1CmdLocalOff	: R_TRIG;
		
		Trig_Pcs1CmdFreqRegOn	: R_TRIG;
		Trig_Pcs1CmdFreqRegOff	: R_TRIG;
		Trig_Pcs1CmdURegOn		: R_TRIG;
		Trig_Pcs1CmdURegOff		: R_TRIG;	
		
	// HVAC
		Trig_Hvac1CmdStart		: R_TRIG;
		Trig_Hvac1CmdStop		: R_TRIG;
		Trig_Hvac2CmdStart		: R_TRIG;
		Trig_Hvac2CmdStop		: R_TRIG;
	
	// PCS1
		bPcs1GridFormer			: BOOL;
		bPcs1GridFeeder			: BOOL;
		bPcs1StartOn			: BOOL;
		bPcs1StartOff			: BOOL;
		bPcs1StopOn				: BOOL;
		bPcs1StopOff			: BOOL;
		bPcs1SoftStopOn			: BOOL;
		bPcs1SoftStopOff		: BOOL;
		bPcs1CmdPOn				: BOOL;
		bPcs1CmdPOff			: BOOL;
		bPcs1CmdQOn				: BOOL;
		bPcs1CmdQOff			: BOOL;	
		bPcs1CmdFreqRegOn		: BOOL;
		bPcs1CmdFreqRegOff		: BOOL;
		bPcs1CmdURegOn			: BOOL;
		bPcs1CmdURegOff			: BOOL;	
		bPcs1CmdLocalOn			: BOOL;
		bPcs1CmdLocalOff		: BOOL;
		bBat1CmdEnable			: BOOL;
		bBat2CmdEnable			: BOOL;
		
		wSystemBMS_Enable		: WORD;
		
	// HVAC
		bHvac1CmdStart			: BOOL;
		bHvac1CmdStop			: BOOL;
		bHvac2CmdStart			: BOOL;
		bHvac2CmdStop			: BOOL;
	
	// PCS1 
		PCS1_SetptP				: REAL;
		PCS1_SetptQ				: REAL;
		PCS1_SetptF				: REAL;
		PCS1_SetptU				: REAL;
		
	// PCS1
		bChange_Pcs1_StptP		: BOOL;
		bChange_Pcs1_StptQ		: BOOL;
		bChange_Pcs1_StptF		: BOOL;
		bChange_Pcs1_StptU		: BOOL;
		bReset_Pcs1				: BOOL;
	
	BBMS1_OpenDC			: BOOL;
	BBMS1_CloseDC			: BOOL;
	BBMS1_Reset				: BOOL;
	
	// Watchdog display 
	
	PCS1_AlarmsStruct		: ARRAY[1..75] OF ST_ValuesAlarms;
	SBMS1_AlarmStruct		: ARRAY[1..60] OF ST_ValuesAlarms;
	StateInv_Local			: STRING;
	HMI_NamePcsEss					: ARRAY[1..CstNbBat_ESS_G*CstNbESS_G] OF STRING(255);
	AX_MailAddr						: ARRAY[1..CstNbUser] OF STRING(255);	//Contient tous les numéros des utilisateurs
	KK: INT;
	LL: INT;
	bPcs1CmdQ: INT;
END_VAR

FOR kk := 1 TO CstNbESS_G DO
	FOR LL := 1 TO CstNbBat_ESS_G DO
		HMI_NamePcsEss[(KK-1)*CstNbBat_ESS_G + LL] := concat('ESS', CONCAT(INT_TO_STRING(KK), concat(' - BAT', INT_TO_STRING(LL))));
	END_FOR
END_FOR



// Ici, le premier élément est le PCS, on récupère le diviseur
ID_ESS_Displayed := DINT_TO_UINT(TRUNC((IN_NumSystemSelected-1) / ParamNbSystemESS))+ 1;
ID_PCS_ESS_Displayed := ((IN_NumSystemSelected-1) MOD CstNbPcs_ESS_G) + 1;
ID_BAT_ESS_Displayed := ((IN_NumSystemSelected-1) MOD CstNbBat_ESS_G) + 1;
ID_PowerCol_PCS_Displayed := (((IN_NumSystemSelected-1) MOD CstNbBat_ESS_G) + 1);


HMI.BMS_Display 		:= AX_ESS[ID_ESS_Displayed].AX_BAT[ID_BAT_ESS_Displayed].MesDataExd;
HMI.PCS_Display			:= AX_ESS[ID_ESS_Displayed].AX_PCS[ID_PCS_ESS_Displayed].MesDataExd;


HMI.ESS_Display 		:= AX_ESS[ID_ESS_Displayed].MesDataExd;



(*
COMMANDS - UNCOMMENT FOR THEM TO WORK
// PCS1 
	IF bChange_Pcs1_StptP THEN 
		bChange_Pcs1_StptP := FALSE;
		OpcUa.AllvalueW.SetptP_PCS[ID_ESS_Displayed][ID_PCS_ESS_Displayed] := PCS1_SetptP;
	END_IF
	IF bChange_Pcs1_StptQ THEN 
		bChange_Pcs1_StptQ := FALSE;
		OpcUa.AllvalueW.SetptQ_PCS[ID_ESS_Displayed][ID_PCS_ESS_Displayed] := PCS1_SetptQ;
	END_IF
	
	OpcUa.AllDataWPulse.CmdLocal_PCS[ID_ESS_Displayed][ID_PCS_ESS_Displayed] := Trig_Pcs1CmdLocalOff.Q;

	IF bPcs1StartOn THEN
		bPcs1StartOn := FALSE;
		OpcUa.AllDataWPulse.CmdStart_PCS[ID_ESS_Displayed][ID_PCS_ESS_Displayed] := TRUE;
	END_IF
	IF bPcs1StopOn THEN
		bPcs1StopOn := FALSE;
		OpcUa.AllDataWPulse.CmdStop_PCS[ID_ESS_Displayed][ID_PCS_ESS_Displayed] := TRUE;
	END_IF
	IF bPcs1SoftStopOn THEN
		bPcs1SoftStopOn := FALSE;
		OpcUa.AllDataWPulse.CmdStandby_PCS[ID_ESS_Displayed][ID_PCS_ESS_Displayed] := TRUE;
	END_IF
	IF bPcs1CmdLocalOn THEN
		bPcs1CmdLocalOn := FALSE;
		OpcUa.AllDataWPulse.CmdLocal_PCS[ID_ESS_Displayed][ID_PCS_ESS_Displayed] := TRUE;
	END_IF
	IF bReset_Pcs1 THEN
		bReset_Pcs1 := FALSE;
		OpcUa.AllDataWPulse.CmdReset_PCS[ID_ESS_Displayed][ID_PCS_ESS_Displayed] := TRUE;
	END_IF

// BMS
	IF BBMS1_CloseDC THEN
		BBMS1_CloseDC := FALSE;
		OpcUa.AllDataWPulse.CmdCloseDc_BAT[ID_ESS_Displayed][ID_BAT_ESS_Displayed] := TRUE;
	END_IF	
	IF BBMS1_OpenDC THEN
		BBMS1_OpenDC := FALSE;
		OpcUa.AllDataWPulse.CmdOpenDc_BAT[ID_ESS_Displayed][ID_BAT_ESS_Displayed] := TRUE;
	END_IF	
	IF BBMS1_Reset THEN
		BBMS1_Reset := FALSE;
		OpcUa.AllDataWPulse.CmdReset_BAT[ID_ESS_Displayed][ID_BAT_ESS_Displayed] := TRUE;
	END_IF	
*)
	
	
// Display bars
	CASE BarDisplay_ID OF
		1:
			BarDisplay_Min := 0;
			BarDisplay_Max := 100;
		2: 
			BarDisplay_Min := -1400;
			BarDisplay_Max := 1400;
		3:
			BarDisplay_Min := 0;
			BarDisplay_Max := 1100;
		4:	
			BarDisplay_Min := 0;
			BarDisplay_Max := 100;
	END_CASE




// Affichage des alarmes
StateInv_Local := SEL(HMI.PCS_Display.MesData.OUT_CmdPcsLocal, 'Remote', 'Local');
//StateInv := concat(PCS_StateInv[AX_ESS[ID_ESS_Displayed].AX_PCS[ID_PCS_ESS_Displayed].MesDataExd.MesData.MesIDState],concat(' - ', StateInv_Local)); 

FOR KK := 57 + 10 * (NumEssDisplayed - 1) TO 66 + 10 * (NumEssDisplayed - 1) DO
	FOR LL := 0 TO 15 DO
		PCS1_AlarmsStruct[(KK-57)*16 + LL+1] := FUN_Alarms.AX_Journal[KK][LL];
	END_FOR
END_FOR


CASE HMI.PCS_Display.MesData.MesID_State_Inv OF 
	973:
		StateInv := '-';
	1787:
		StateInv := 'Init';
	381:
		StateInv := 'Stop';
	1392:
		StateInv := 'Error';
	3522:
		StateInv := 'Update';
	3523:
		StateInv := 'Reset';
	1394:
		StateInv := 'WaitAC';
	3524:
		StateInv := 'ConnectAC';
	1393:
		StateInv := 'WaitDC';
	3525:
		StateInv := 'ConnectDC';
	3526:
		StateInv := 'GridFeed';
	21429:
		StateInv := 'GridForm';
	21584:
		StateInv := 'ActRampUp';
	3527:
		StateInv := 'FRT';
	3528:
		StateInv := 'Standby';
	3529:
		StateInv := 'QonDemand';
	3530:
		StateInv := 'RampDown';
	375:
		StateInv := 'Selftest';
	3533:
		StateInv := 'IOTest';
	ELSE
		StateInv := 'Unknown';
END_CASE

END_PROGRAM

// ---- 04_Application/HMI/SPP/SPP_HMI.TcPOU
PROGRAM SPP_HMI
VAR
	AX_INV_Eday 		: ARRAY[1..CstNbInv_PTR_G] OF REAL;
	AX_INV_P	 		: ARRAY[1..CstNbInv_PTR_G] OF REAL;
	
	HMI_NameInvPtr		: ARRAY[1..CstNbInv_PTR_G] OF STRING(255);
	IN_NumSppDisplayed	: UINT := 1;
	
	KK, LL : UINT;
	ID_PTR_Displayed: UINT;
	ID_INV_PTR_Displayed: UINT;
END_VAR




// Ici, le premier élément est le PCS, on récupère le diviseur
ID_PTR_Displayed := DINT_TO_UINT(TRUNC((IN_NumSppDisplayed-1)/CstNbInv_PTR_G))+ 1;
ID_INV_PTR_Displayed := ((IN_NumSppDisplayed-1) MOD CstNbInv_PTR_G) + 1;

FOR LL := 1 TO CstNbInv_PTR_G DO
	HMI_NameInvPtr[LL] := concat('PTR', CONCAT(INT_TO_STRING(ID_PTR_Displayed), concat(' - INV', INT_TO_STRING(LL))));
END_FOR

HMI.PTR_Display 		:= AX_PTR[ID_PTR_Displayed].MesDataExd;
HMI.INV_Display			:= AX_PTR[ID_PTR_Displayed].AX_INV[ID_INV_PTR_Displayed].MesDataExd;

END_PROGRAM

// ---- 00_FunctionsBlocks/Beckhoff/DataProcessing/SavePersistent.TcPOU
PROGRAM SavePersistent
///////////////////
// Save persistent data regularly
///////////////////
VAR
	FB_WritePersistentData : WritePersistentData  ;
	
	LTP2: TP;
	ClockPersistent: BOOL;
END_VAR

// WRITING CLOCK //
	LTP2(IN:=NOT LTP2.Q , PT:= T#1M);
	ClockPersistent := LTP2.Q;

FB_WritePersistentData(
						NETID:='', 
						PORT:= 851 ,
						START :=  ClockPersistent AND NOT FB_WritePersistentData.BUSY , 
						TMOUT := T#10S ) ;

END_PROGRAM

// ---- 00_FunctionsBlocks/Beckhoff/Communication/Mail/FUN_SendMail.TcPOU
PROGRAM FUN_SendMail
////////////////// 
// Send Alarms by mails. 
//////////////////

VAR_INPUT 
	
	IN_Reset_OPC					: BOOL;					// Reset Mail server and alarms. 
	IN_ChangePhoneMailInfos_OPC		: BOOL;					// Change users Info (mails, name, Lvl, ... ) 
	FIFO							: FB_DBDatasetFifo;		// Buffer of the alarmes). 
	
	MesData			: ServerMail;
	
END_VAR

VAR_OUTPUT
	OUT_Error						: BOOL ; // Send Email Error 
	OUT_Completed					: BOOL;		// Juste un trig pour dire que c'est fini. Written by the SMTP.Exe
	OUT_NbMailSent 					: UINT;	// Number of mail being sent. 
	
END_VAR

VAR PERSISTENT
	
	AX_MailAddr						: ARRAY[1..CstNbUser] OF STRING(255);	//Contient tous les numéros des utilisateurs
	AX_Subscribed					: ARRAY[1..CstNbUser] OF BOOL		;	// List of subscription. 
	AX_NomUtili						: ARRAY[1..CstNbUser] OF STRING(50)	;	// List of user names. 
	AX_User_LVL						: ARRAY[1..CstNbUser] OF WORD;			//Contient tous les niveau d'adhésion des utilisateurs.
	
END_VAR

VAR_INPUT PERSISTENT
	
	ParamTempoRetry					: TIME := T#1M;  (* (s) Tempo before send email retry *) 
	
END_VAR

VAR

	// M_AlarmManager 

	RS_AlarmDestinator		: RS;
	RS_AlarmSendMailFail	: RS;
	
	// M_Write Param	
	bAlarmNoDestinator		: BOOL;
	bSendMail				: BOOL;
	
	Body					: T_MaxString;
	MailAddr				: T_MaxString;
	MesTimeStamp			: STRING(17);	
	CalTimeStamp			: STRING(255);
	
	//M_OPC
	Trig_OPC				: R_TRIG;
	RS_OPC					: RS;
	Trig_Reset				: R_TRIG;

	KK						: UINT;
	NbDest					: INT;
	TON_Retry				: TON;
	Old_Count				: UDINT;
	R_TRIG_Retry			: R_TRIG;

// New Sender
	NewSender 				: NT_StartProcess;
	
END_VAR

M_AlarmManager();
M_OPC();
M_Evaluate();

IF IN_Reset_OPC THEN
	M_Reset();
END_IF
TON_Retry(IN := Old_Count = fifo.nCount AND NOT R_TRIG_Retry.Q, pt := ParamTempoRetry);

R_TRIG_Retry(clk := TON_Retry.Q);
IF old_count <> fifo.nCount THEN
	Old_Count := fifo.nCount;
END_IF

fifo.A_Get();	// Get the next alarm to send. 

MesTimeStamp := CONCAT(REPLACE(STR1:= left(str := FIFO.Out.TimeStamp_Act, 16), STR2 := ' ', L := 1, P := 11), ' ') ;
ReplaceAll( In_StringTosearch := MesTimeStamp, In_StringToFind := '/', IN_StringToReplace := '-', OUT_StringToSearch => CalTimeStamp);

Body := concat(left(FIFO.Out.Message, 125),SEL(FIFO.Out.Value, ' : Desactive"',' : Active"')) ; 
Body := concat( STR1:= UINT_TO_STRING(FIFO.Out.ID) , STR2:= concat(STR1:=' ,' , STR2:=Body )) ; 
Body := concat( STR1:= 'ID:' , STR2:=Body ) ; 
Body := concat('"', Concat(CalTimeStamp,Body));


MailAddr := '"';
NbDest := 0;
FOR KK := 1 TO CstNbUser DO
	IF AX_Subscribed[KK] AND AX_MailAddr[KK] <> '' AND (AX_User_LVL[KK] AND Fifo.out.Alarms_LVL)>0 THEN		// If user is subscribed to this alarm, add his mail adress to the list. 
		IF MailAddr = '"' THEN
			MailAddr := concat('"', AX_MailAddr[KK]);	// Initialize first sender. 
		END_IF
		NbDest := NbDest + 1;
	END_IF
END_FOR

IF NbDest >0 THEN
	IF NbDest>1 THEN
		FOR KK := 1 TO CstNbUser DO
			IF AX_Subscribed[KK] AND MailAddr <> AX_MailAddr[KK] AND (AX_User_LVL[KK] AND Fifo.out.Alarms_LVL)>0 THEN
				MailAddr := concat(concat(MailAddr, ', '), AX_MailAddr[KK]);		// append other mail adress if several users subsribed to this alarm. 
			END_IF
		END_FOR
	END_IF
	MailAddr := concat(MailAddr, '"');
	bSendMail := TRUE;
	bAlarmNoDestinator	:= FALSE;
ELSE 
	bAlarmNoDestinator	:= TRUE;
	bSendMail 			:= FALSE;
	FIFO.A_Remove();	// remove alarm from FIFO if no destinator to avoid blocking the process
END_IF	

IF fifo.nCount = 0 THEN
	bSendMail := FALSE;
END_IF

IF OUT_Completed THEN 
	OUT_Completed := FALSE;
	OUT_NbMailSent := OUT_NbMailSent + 1;

	bSendMail := FALSE;
	FIFO.A_Remove();
END_IF	

IF OUT_NbMailSent > 30000 THEN
	OUT_NbMailSent := 0;
END_IF

METHOD M_AlarmManager
VAR
	
	FB_AlarmCodeManager : FB_AlarmCodeManager;

END_VAR
// Gestion des alarmes internes au code

RS_AlarmDestinator(SET:= bAlarmNoDestinator , RESET1:= IN_Reset_OPC ) ; 
RS_AlarmSendMailFail(set := OUT_Error, reset1 := IN_Reset_OPC);

FB_AlarmCodeManager
(
	bAlarm1 := RS_AlarmDestinator.Q1,			// No recipient for at least one alarm
	bAlarm2 := FALSE,						// 
	bAlarm3 := RS_AlarmSendMailFail.Q1,			// Execution of NewSender.exe did not work.  
	bAlarm4 := FIFO.bOverwrite,					// Fifo Overflow
	bAlarm5 := FALSE,							//
	bAlarm6 := FALSE,    						//
	bAlarm7 := FALSE,    						//
	bAlarm8 := FALSE,    						//
	bAlarm9 := FALSE,    						//
	bAlarm10 :=FALSE,   						//
	bAlarm11 :=FALSE,   						//
	bAlarm12 :=FALSE,   						//
	bAlarm13 :=FALSE,   						//
	bAlarm14 :=FALSE,   						//
	bAlarm15 :=FALSE,							//	
	wAlarmCode =>MesData.MesAlarmCode
);
END_METHOD

METHOD M_Evaluate
VAR 
END_VAR

Mesdata.AX_MailAddr		:= AX_MailAddr			;
Mesdata.AX_Subscribed	:= AX_Subscribed	    ;
MesData.AX_NomUtili		:= AX_NomUtili		    ;
MesData.OUT_NbMailSent	:= OUT_NbMailSent		;
MesData.AX_UserLVL		:= AX_User_LVL		    ;
END_METHOD

METHOD M_Init : BOOL
VAR_INPUT
END_VAR
END_METHOD

METHOD M_OPC : BOOL
VAR

END_VAR
Trig_OPC(CLK := IN_ChangePhoneMailInfos_OPC);
RS_OPC(SET:= Trig_OPC.Q);

//TrigRestartService(CLK := IN_Restart_Service_OPC);
//FUN_RestartStunnel(IN_Start := TrigRestartService.Q, IN_Directory := IN_Directory);


IF RS_OPC.Q1 THEN
	// Numéro de téléphone
	AX_MailAddr := OpcUa.AllValueW.AX_MailAddr_OPC;
	
	// Nom d'utilisateur
	AX_NomUtili	:= OpcUa.AllValueW.AX_NamesUsers_OPC;
	
	// User LVL . 
	AX_User_LVL := OpcUa.AllValueW.AX_UserLVL;
	
	// Mise a jour de la liste des subscribed
	AX_Subscribed := OpcUa.AllValueW.AX_SubscribedMail_OPC;

	RS_OPC(RESET1:= TRUE);
	RS_OPC(Reset1 := FALSE);
END_IF

Trig_Reset(CLK := IN_Reset_OPC);
IN_Reset_OPC := Trig_Reset.Q;
END_METHOD

METHOD M_Reset : BOOL
VAR_INPUT
END_VAR
VAR
	

END_VAR
FIFO.A_Reset();
IN_Reset_OPC 			:= FALSE;
bAlarmNoDestinator 		:= FALSE ;	
bSendMail				:= FALSE;
END_METHOD

END_PROGRAM

// ---- 00_FunctionsBlocks/Beckhoff/Database/InfluxDb/InfluxDb_AlarmsManagement.TcPOU
PROGRAM InfluxDb_AlarmsManagement

VAR_INPUT
	IN_FIFO										: FB_DBDatasetFifo;
	IN_Reset									: BOOL;
	//MesDataExd								: LoggerInfluxDb;
END_VAR

VAR
	// M_Init
   		bInit 									: BOOL;
	// Reset                					
		Trig_Reset								: R_TRIG;
	// Interface values
		bGet: BOOL;
		bRem: BOOL;
		Out_Alarms 				: ST_ValuesAlarms;
		Out_Alarms_Null 		: ST_ValuesAlarms;
END_VAR

IF NOT bInit THEN
	M_Init();
END_IF

Trig_Reset(CLK := IN_Reset OR CmdClearFault_G);
IF Trig_Reset.Q THEN
	IN_Reset := FALSE;
	IN_FIFO.A_Reset();
	Out_Alarms := Out_Alarms_Null;
END_IF

IF bRem THEN
	bRem := FALSE;
	IN_FIFO.A_Remove();
	Out_Alarms := Out_Alarms_Null;
END_IF

IF bGet THEN
	bGet := FALSE;
	IN_FIFO.A_Get();
	Out_Alarms := IN_FIFO.Out;
END_IF

METHOD M_Init : BOOL
VAR_INPUT
END_VAR
//Initialisation BUFFER
	//Buffer pour la lecture des sms
	//IN_FIFO.A_Reset();
	//IN_FIFO.A_Add();
	//IN_FIFO.A_Get();
	//IN_FIFO.A_Remove();
	
	IN_FIFO.In.Message :=  'Code Activation';
	IN_FIFO.IN.TimeStamp_Act := SYSTEMTIME_TO_STRING(CalLocalTimeStruct);
	IN_FIFO.A_Add();
	bInit := TRUE;
END_METHOD

END_PROGRAM

// ---- 04_Application/ALARM/Redundancy.TcPOU
PROGRAM Redundancy
///////////////////
// Exchange redundant data : parameters , bistable functions, setpoints , PID values ( integer ) 
///////////////////
VAR_INPUT PERSISTENT
	// Parameters of the Object (instance specific) 
		ParamTimeout					: TIME  := T#1S ;				// (Time) Timeout for modbus reading
		ParamTempoImpulsion2			: TIME := T#500MS ; 			// ADS Clock Read Time < Timeout
		ParamNbSignalRedundancy			: UINT := 233 ;					// Number of signals defined for the redundancy
END_VAR

VAR
	Address							: ARRAY[1..CstNbRedundantVariableMax_G] OF PVOID ;		
	SignalName						: ARRAY[1..CstNbRedundantVariableMax_G] OF STRING ;		
	PLC_ReadSymInfoByName	        : ARRAY[1..CstNbRedundantVariableMax_G] OF  PLC_ReadSymInfoByName	;
	ReadAds		                  	: ARRAY[1..CstNbRedundantVariableMax_G] OF ADSREADEX;

	
	// ClockRead
	TP1 						: TP ; 
	R_TRIG_Read					: R_TRIG ; 	
	ClockRead					: BOOL ; 		
	
	nPort				  		: UINT := 851;					    // (NA) ADS device Port
	bInit						: BOOL := TRUE ;	
	
END_VAR

METHOD M_GetRedundancyData
VAR_INPUT
END_VAR
END_METHOD

METHOD M_Init : BOOL
VAR_INPUT
END_VAR
END_METHOD

METHOD M_ReadRedundancyData 
VAR
	CP_Read  		: ARRAY[1..CstNbRedundantVariableMax_G] OF BOOL ; 
	
	KK				: UINT;
	JJ				: UINT;
	bCopyCP			: BOOL;	// force CP to false . 
END_VAR

// ClockRead 
TP1(IN:= NOT TP1.Q,PT:=ParamTempoImpulsion2);
R_TRIG_Read(CLK:=TP1.Q,Q=>ClockRead);

FOR KK:= 1 TO ParamNbSignalRedundancy DO 
	// Get INfos 
	PLC_ReadSymInfoByName[KK](NETid := CstNetAmsId_Slave, Port:=nPort,Symname:=SignalName[KK], Start:= CalLocalTimeStruct.wSecond=KK OR bInit,TMOUT:= T#5S) ;
	CP_Read[KK] := ClockRead  AND NOT (PLC_ReadSymInfoByName[KK].SYMINFO.idxOffset=0) AND NOT PLC_ReadSymInfoByName[KK].ERR AND NOT ReadAds[KK].BUSY  ; 


	// Read signal 
	ReadAds[KK](NETID:=CstNetAmsId_Slave,
				   PORT:=nPort,
				   IDXGRP:=	PLC_ReadSymInfoByName[KK].SYMINFO.idxGroup,
				   IDXOFFS:=PLC_ReadSymInfoByName[KK].SYMINFO.idxOffset,
				   LEN:=PLC_ReadSymInfoByName[KK].SYMINFO.byteSize,
				   READ:=CP_Read[KK],
				   DESTADDR:=Address[KK], 
				   TMOUT:=ParamTimeout);


END_FOR



bInit:= FALSE ;

// For all.MesDataExd.MesData.CalCPRead and Write to False when redundancy is activated 

bCopyCP := FALSE  ; 

(*
	FOR KK:= 1 TO CstNbESs DO 
		FOR JJ:= 1 TO CstNbBank_Ess DO 
			 	MEMCPY(ADR(AX_ESS[KK].AX_Bat[JJ].MesCP_Write  ),ADR(bCopyCP),SIZEOF(bCopyCP));
			 	MEMCPY(ADR(AX_ESS[KK].AX_Bat[JJ].MesCP_Read  ),ADR(bCopyCP),SIZEOF(bCopyCP));
		END_FOR
		FOR JJ:= 1 TO CstNbPcs_Ess DO 
			 	MEMCPY(ADR(AX_ESS[KK].AX_PCS[JJ].MesCP_Write  ),ADR(bCopyCP),SIZEOF(bCopyCP));
			 	MEMCPY(ADR(AX_ESS[KK].AX_PCS[JJ].MesCP_Read  ),ADR(bCopyCP),SIZEOF(bCopyCP));
		END_FOR
		FOR JJ:= 1 TO CstNbHvac_ESS DO 
			 MEMCPY(ADR(AX_ESS[KK].AX_HVAC[JJ].MesCP_Write  ),ADR(bCopyCP),SIZEOF(bCopyCP));
			 MEMCPY(ADR(AX_ESS[KK].AX_HVAC[JJ].MesCP_Read  ),ADR(bCopyCP),SIZEOF(bCopyCP));
		END_FOR
	END_FOR 
	
	 MEMCPY(ADR(A1_SUB_MV.A1_GRID.MesCP_Read  			),ADR(bCopyCP),SIZEOF(A1_SUB_MV.A1_GRID.MesCP_Read  			));
	 MEMCPY(ADR(A1_SUB_MV.A1_PM_Aux.MesCP_Read          ),ADR(bCopyCP),SIZEOF(A1_SUB_MV.A1_PM_Aux.MesCP_Read          ) );
	 MEMCPY(ADR(A1_SUB_MV.A1_ProtectionRelay_ImBess1 .MesCP_Read   ),ADR(bCopyCP),SIZEOF(A1_SUB_MV.A1_ProtectionRelay_ImBess1 .MesCP_Read   ) );
	 MEMCPY(ADR(A1_SUB_MV.A1_ProtectionRelay_ImBess2 .MesCP_Read   ),ADR(bCopyCP),SIZEOF(A1_SUB_MV.A1_ProtectionRelay_ImBess2 .MesCP_Read   ) );
	 MEMCPY(ADR(A1_SUB_MV.A1_ProtectionRelay_ImBess3 .MesCP_Read   ),ADR(bCopyCP),SIZEOF(A1_SUB_MV.A1_ProtectionRelay_ImBess3 .MesCP_Read   ) );
	 MEMCPY(ADR(A1_SUB_MV.A1_ProtectionRelay_ImBess4 .MesCP_Read   ),ADR(bCopyCP),SIZEOF(A1_SUB_MV.A1_ProtectionRelay_ImBess4 .MesCP_Read   ) );
	 MEMCPY(ADR(A1_SUB_MV.A1_ProtectionRelay_ImBess5 .MesCP_Read   ),ADR(bCopyCP),SIZEOF(A1_SUB_MV.A1_ProtectionRelay_ImBess5 .MesCP_Read   ) );
	 MEMCPY(ADR(A1_SUB_MV.A1_ProtectionRelay_ImBess6 .MesCP_Read   ),ADR(bCopyCP),SIZEOF(A1_SUB_MV.A1_ProtectionRelay_ImBess6 .MesCP_Read   ) );
	 MEMCPY(ADR(A1_SUB_MV.A1_UPS_SUB_MV.MesCP_Read        ),ADR(bCopyCP),SIZEOF(A1_SUB_MV.A1_UPS_SUB_MV.MesCP_Read        ) );
	
	FOR KK:=1 TO 2 DO 
		MEMCPY(ADR(A1_SUB_MV.AX_PM[KK].MesCP_Read  ),ADR(bCopyCP),SIZEOF(A1_SUB_MV.AX_PM[KK].MesCP_Read ));
		
	END_FOR
// 	
	*)
END_METHOD

END_PROGRAM

// ---- 04_Application/BDD/FUN_Write_CSV.TcPOU
PROGRAM FUN_Write_CSV

VAR_INPUT
 InDirectory             : T_MaxString;
AX_Variables            : ARRAY [1..500] OF ST_ValuesWrite;
    WriteValue          : FB_Write_CSV;
END_VAR


AX_Variables[ 1].Address := ADR(A1_SUBMV.MesDataExd.MesData.MesU);AX_Variables[ 1].Description :='SUBMV:// (V) Mean Phase to Phase grid voltage';
AX_Variables[ 1].Size:= SIZEOF(A1_SUBMV.MesDataExd.MesData.MesU);AX_Variables[ 1].sampling := 60000;
AX_Variables[ 2].Address := ADR(A1_SUBMV.MesDataExd.MesData.MesFreq);AX_Variables[ 2].Description :='SUBMV:// (Hz) Grid Frequency';
AX_Variables[ 2].Size:= SIZEOF(A1_SUBMV.MesDataExd.MesData.MesFreq);AX_Variables[ 2].sampling := 60000;
AX_Variables[ 3].Address := ADR(A1_SUBMV.MesDataExd.MesData.MesPsol);AX_Variables[ 3].Description :='SUBMV:// (kW) Total Solar Active Power';
AX_Variables[ 3].Size:= SIZEOF(A1_SUBMV.MesDataExd.MesData.MesPsol);AX_Variables[ 3].sampling := 60000;

WriteValue(InDirectory := InDirectory, ParamNbColumns := 3,AX_StructureValues := AX_Variables);

END_PROGRAM

// ---- 00_FunctionsBlocks/Beckhoff/DataProcessing/WriteFile/FB_Write_CSV.TcPOU
FUNCTION_BLOCK FB_Write_CSV
VAR_INPUT
	InDirectory 		: T_MaxString;
	AX_StructureValues	: ARRAY[1..500] OF ST_ValuesWrite;
	
	ParamNbColumns		: UINT := 200; 				(* (NA) Number of columns of the file*)
	ParamSeparateur		: STRING := ';';			(* (NA) Separator*)
	ParamDec			: STRING := ',';			(* (NA) ParamDec*)
	ParamExtension		: T_MaxString := '.csv'; 	(* (NA) csv extension *)
	
	
	MesData		: LoggerCSV;
	
END_VAR
VAR_OUTPUT
END_VAR
VAR
	
    CompressFile        : FB_CompressFile;


	bWriteAlarm			: BOOL;						// Writing CSV File failed 
	TON_WritealarmFile	: TON;	
	// Data processing 
	format_string		: FB_FormatString;
	AX_AverageFunctions	: ARRAY[1..1000] OF FB_Average;
	AX_AverageValues	: ARRAY[1..1000] OF REAL;
	LenStringToWrite	: INT;
	
	GetHostName			: FB_GetHostName;
	CalFileName			: STRING;
	CalFileName_Old		: STRING;
	CalDate				: STRING;
	CalDate_Old			: STRING;
	
	//Test existence file 

	bFileOK				: BOOL := TRUE ;
	bDirChange			: BOOL;
	FindFile 			: FB_EnumFindFileEntry ;
	FileInfo			: ST_FindFileEntry;
	
	//Initial File creation 
	InitLine			: T_MaxString;
	LastInitLine		: T_MaxString;
	WelcomeMessage 		: T_MaxString := 'Daily rawdata file';
	ForDay				: T_MaxString := 'for day : ';
	ForPlant	 		: T_MaxString := 'for plant : ';
	NewLineVar			: T_MaxString := '$N';
	TimeStampVar		: T_MaxString := 'TimeStamp';
	len_to_write		: INT;
	len_to_add			: INT;
	
	WriteFileInit		: FB_WriteFile;
	WriteFile			: FB_WriteFile;
	MessageInitial		: ARRAY[1..100] OF T_Maxstring;
	MessageInitialNull	: ARRAY[1..100] OF T_Maxstring;
	bInitWrite			: BOOL;
	bInitWriting		: BOOL;
	
	// Write File
	LineToWrite			: ARRAY [1..100] OF  T_Maxstring;
	LineToWrite_Null	: ARRAY [1..100] OF  T_Maxstring;
	ValueToWrite		: T_MaxString;
	TriggerSampling		: R_TRIG;
	
	// General variables
	KK: UINT;
	bInit : BOOL;
	MesTimeStamp : STRING(19);
	

	
END_VAR

M_AlarmManager();
M_DataProcessing ();

IF NOT bInit THEN
	GetHostName(bExecute := FALSE);
	GetHostName(bExecute := TRUE);
	bInit := TRUE;
END_IF

format_string(
	sFormat := 'RAWDATA_%0.2d-%0.2d-%0.2d%s', 
	arg1 := F_WORD(in:=CalLocalTimeStruct.wYear),	arg2 := F_WORD(in:=CalLocalTimeStruct.wMonth),	arg3 := F_WORD(in:=CalLocalTimeStruct.wDay),
	arg4 := F_STRING(in:=ParamExtension),
	sOut => CalFileName
);

format_string(
	sFormat := '%0.2d-%0.2d-%0.2d', 
	arg1 := F_WORD(in:=CalLocalTimeStruct.wYear),	arg2 := F_WORD(in:=CalLocalTimeStruct.wMonth),	arg3 := F_WORD(in:=CalLocalTimeStruct.wDay),
	sOut => CalDate
);

format_string(
	sFormat := '%0.2d-%0.2d-%0.2d %0.2d:%0.2d:%0.2d', 
	arg1 := F_WORD(in:=CalLocalTimeStruct.wYear),	arg2 := F_WORD(in:=CalLocalTimeStruct.wMonth),	arg3 := F_WORD(in:=CalLocalTimeStruct.wDay),
	arg4 := F_WORD(in:=CalLocalTimeStruct.wHour),	arg5 := F_WORD(in:=CalLocalTimeStruct.wMinute),	arg6 := F_WORD(in:=CalLocalTimeStruct.wSecond),
	sOut => MesTimeStamp
);

InitLine := concat(str1:=WelcomeMessage, STR2:= concat(str1:=
	ParamSeparateur, str2:=concat(STR1:=ForDay, STR2:=concat(str1:= ParamSeparateur, STR2:= concat(str1:= 
	CalDate,str2:=concat(str1:= ParamSeparateur, str2 := CONCAT(str1:=
	ForPlant,str2:=Concat(str1:=ParamSeparateur, str2:= CONCAT(str1:= GetHostName.sHostName, str2:=ParamSeparateur)
))))))));

IF InitLine <> LastInitLine OR InitLine = '' OR (NOT FindFile.bError AND NOT bFileOK) THEN
	LastInitLine := InitLine;
	bInitWriting := TRUE;
END_IF
	
IF FUN_CreateDir_CSV.bDirOK THEN
	FindFile
	(
		sNetId := '',
		sPathName := concat(FUN_CreateDir_CSV.AX_DirNames[2],CalFileName),
		eCmd := eEnumCmd_First,
		bExecute := TRUE,
		tTimeout := T#3S,
		stFindFile => FileInfo
	);
	
MesData.TimeCreation 	:= FILETIME_TO_SYSTEMTIME(filetime := FileInfo.creationTime);
MesData.TimeModif	 	:= FILETIME_TO_SYSTEMTIME(filetime := FileInfo.lastWriteTime);
MesData.FileSize  		:= ULARGE_TO_ULINT(in := FileInfo.fileSize);	
	
	IF NOT FindFile.bBusy THEN
		FindFile(bExecute := FALSE);
		bFileOK := MesData.FileSize > 0 ; 
	END_IF
	
	IF FindFile.bError OR  NOT bFileOK THEN
		FUN_CreateDir_CSV(InDirectory := ParamDirBaseStore, RESET2 := TRUE);
	END_IF
	
	IF NOT FindFile.bBusy AND NOT bFileOK AND bInitWriting THEN
		// je réinitialise les longueurs
		len_to_write := 0;
		MessageInitial := MessageInitialNull;
		MEMCPY(destAddr := ADR(MessageInitial)+len_to_write, srcAddr := ADR(InitLine), n := len(InitLine));
		len_to_add := len(InitLine);			len_to_write := len_to_write + len_to_add;
		
		MEMCPY(destAddr := ADR(MessageInitial)+len_to_write, srcAddr := ADR(NewLineVar), n := len(NewLineVar));
		len_to_add := len(NewLineVar);			len_to_write := len_to_write + len_to_add;
		
		MEMCPY(destAddr := ADR(MessageInitial)+len_to_write, srcAddr := ADR(TimeStampVar), n := len(TimeStampVar));
		len_to_add := len(TimeStampVar);		len_to_write := len_to_write + len_to_add;
		
		MEMCPY(destAddr := ADR(MessageInitial)+len_to_write, srcAddr := ADR(ParamSeparateur), n := len(ParamSeparateur));
		len_to_add := len(ParamSeparateur);		len_to_write := len_to_write + len_to_add;
		
		FOR KK := 1 TO ParamNbColumns DO
			MEMCPY(destAddr := ADR(MessageInitial)+len_to_write, srcAddr := ADR(AX_StructureValues[KK].Description), n := len(AX_StructureValues[KK].Description));
			len_to_add := len(AX_StructureValues[KK].Description);			len_to_write := len_to_write + len_to_add;
			
			MEMCPY(destAddr := ADR(MessageInitial)+len_to_write, srcAddr := ADR(ParamSeparateur), n := len(ParamSeparateur));
			len_to_add := len(ParamSeparateur);								len_to_write := len_to_write + len_to_add;
		END_FOR
		
		MEMCPY(destAddr := ADR(MessageInitial)+len_to_write, srcAddr := ADR(NewLineVar), n := len(NewLineVar));
		len_to_add := len(NewLineVar);			len_to_write := len_to_write + len_to_add;
		
		WriteFileInit
		(
			InStart := TRUE,
			InDirFile := concat(FUN_CreateDir_CSV.AX_DirNames[2], CalFileName),
			InAmsId := '', 
			InPMessage := ADR(MessageInitial),
			InLMessage := len_to_write
		);
		
		IF WriteFileInit.OutCompleted OR bFileOK THEN
			WriteFileInit(InStart := FALSE);
		END_IF
	END_IF
	
	
	// Write file on SampleRate
	
	TriggerSampling(clk := CalLocalTimeStruct.wSecond = 10);

	IF bFileOK AND MesData.FileSize < 100000000  THEN
		bInitWriting := FALSE;
		len_to_write := 0;
		LineToWrite := LineToWrite_Null;
		MEMCPY(destAddr := ADR(LineToWrite)+len_to_write, srcAddr := ADR(MesTimeStamp), n := len(MesTimeStamp));
		len_to_add := len(MesTimeStamp);		len_to_write := len_to_write + len_to_add;
		
		MEMCPY(destAddr := ADR(LineToWrite)+len_to_write, srcAddr := ADR(ParamSeparateur), n := len(ParamSeparateur));
		len_to_add := len(ParamSeparateur);		len_to_write := len_to_write + len_to_add;
		
		FOR KK := 1 TO ParamNbColumns DO
			ReplaceAll(IN_StringToSearch := REAL_TO_STRING(AX_AverageValues[KK]), IN_StringToFind := '.', IN_StringToReplace := ParamDec, OUT_StringToSearch => ValueToWrite);
			//ValueToWrite := REAL_TO_STRING(AX_AverageValues[KK]);
			MEMCPY(destAddr := ADR(LineToWrite)+len_to_write, srcAddr := ADR(ValueToWrite), n := len(ValueToWrite));
			len_to_add := len(ValueToWrite);	len_to_write := len_to_write + len_to_add;
			
			MEMCPY(destAddr := ADR(LineToWrite)+len_to_write, srcAddr := ADR(ParamSeparateur), n := len(ParamSeparateur));
			len_to_add := len(ParamSeparateur);	len_to_write := len_to_write + len_to_add;
		END_FOR
		MEMCPY(destAddr := ADR(LineToWrite)+len_to_write, srcAddr := ADR(NewLineVar), n := len(NewLineVar));
		len_to_add := len(NewLineVar);			len_to_write := len_to_write + len_to_add;
		
		WriteFile
		(
			InStart := TriggerSampling.Q,
			InDirFile := concat(FUN_CreateDir_CSV.AX_DirNames[2], CalFileName),
			InAmsId := '', 
			InpMessage := ADR(LineToWrite),
			InLMessage := len_to_write
		);
		
		IF NOT WriteFile.OutBusy AND NOT WriteFile.OutError AND WriteFile.OutCompleted THEN
			// File has been writen successfully
			bWriteAlarm	:= FALSE ;
		ELSIF WriteFile.OutError THEN 
			// In case of writing error, try again to write the alarm. 
			bWriteAlarm	:= TRUE ;
		
		END_IF		
		
	END_IF

END_IF

CompressFile(IN_Directory := InDirectory);

METHOD M_AlarmManager
VAR

	FB_AlarmCodeManager			: FB_AlarmCodeManager ;

END_VAR
TON_WritealarmFile(IN:= NOT bFileOK  , PT:= T#10S  ) ;

// ALARM CODE //
	FB_AlarmCodeManager(
		bAlarm1			:= bWriteAlarm	  ,				// Write CSV Alarm
		bAlarm2			:= FALSE   ,					// 
		bAlarm3			:= TON_WritealarmFile.Q   ,		// Can not create CSV Alarm file 
		bAlarm4			:= FALSE	 ,					//
		bAlarm5			:= FALSE	,					// 
		bAlarm6			:= FALSE,									//
		bAlarm7			:= FALSE,                                   //
		bAlarm8			:= FALSE,                                   //
		bAlarm9			:= FALSE,                                   //
		bAlarm10		:= FALSE,                                   //
		bAlarm11		:= FALSE,									//
		bAlarm12		:= FALSE,                                   //
		bAlarm13		:= FALSE,                                   //
		bAlarm14		:= FALSE,                                   //
		bAlarm15		:= FALSE,                                   //
		wAlarmCode		=>MesData.MesAlarmCode);
END_METHOD

METHOD M_DataProcessing : BOOL
VAR
		
	KK : UINT;
END_VAR
FOR KK := 1 TO ParamNbColumns DO 
	IF AX_StructureValues[KK].Address <> 0 THEN 	
		AX_AverageFunctions[KK](ValueIn := AX_StructureValues[KK].Address^, WindowDuration := AX_StructureValues[KK].Sampling, CycleTime := CstCycleTime_Annex, ValueOut=> AX_AverageValues[KK]);	
	ELSIF AX_StructureValues[KK].AddressLR <> 0 THEN 	
		AX_AverageFunctions[KK](ValueIn := AX_StructureValues[KK].AddressLR^, WindowDuration := AX_StructureValues[KK].Sampling, CycleTime := CstCycleTime_Annex, ValueOut=> AX_AverageValues[KK]);	
	ELSIF AX_StructureValues[KK].AddressUL <> 0 THEN 	
		AX_AverageFunctions[KK](ValueIn := AX_StructureValues[KK].AddressUL^, WindowDuration := AX_StructureValues[KK].Sampling, CycleTime := CstCycleTime_Annex, ValueOut=> AX_AverageValues[KK]);	
	ELSIF AX_StructureValues[KK].AddressUI <> 0 THEN
		AX_AverageFunctions[KK](ValueIn := AX_StructureValues[KK].AddressUI^, WindowDuration := AX_StructureValues[KK].Sampling, CycleTime := CstCycleTime_Annex, ValueOut=> AX_AverageValues[KK]);			
	ELSE
		AX_AverageValues[KK] := 0;
	END_IF
END_FOR
END_METHOD

END_FUNCTION_BLOCK

// ---- 00_FunctionsBlocks/Beckhoff/DataProcessing/Compress/FB_CompressFile.TcPOU
FUNCTION_BLOCK FB_CompressFile
// FB to Compress all files of the directory. 
VAR_INPUT
	IN_Directory			: T_MaxString; // directory of the file to compress
END_VAR
VAR_OUTPUT
END_VAR
VAR
	StartProcess 			: NT_StartProcess;
	bTest 					: BOOL;
	TrigJour				: R_TRIG;
	RsJour					: RS;
	DirAlarms				: T_MaxString;
	DirRawdata				: T_MaxString;
	TimeStructYesterday		: TIMESTRUCT;
END_VAR


TrigJour(CLK := CalLocalTimeStruct.wHour =0);
RsJour(SET := TrigJour.Q);

TimeStructYesterday := DT_TO_SYSTEMTIME( SYSTEMTIME_TO_DT (CalLocalTimeStruct) - T#1D);

IF RsJour.Q1 THEN
	DirAlarms := CONCAT(STR1 := CONCAT(STR1 := CONCAT(STR1 := CONCAT(STR1 := CONCAT(STR1 := CONCAT(STR1 := CONCAT(STR1 := CONCAT(STR1 := CONCAT(STR1 := Concat(STR1 := Concat(STR1 := IN_Directory, STR2 := WORD_TO_STRING(TimeStructYesterday.wYear)), STR2 := '\'), STR2 := WORD_TO_STRING(TimeStructYesterday.wMonth)), STR2 := '\'), STR2:='ALARMS_'), STR2:= WORD_TO_STRING(TimeStructYesterday.wYear)), STR2:='-'),STR2:=WORD_TO_STRING(TimeStructYesterday.wMonth)),STR2:='-'),STR2:=WORD_TO_STRING(TimeStructYesterday.wDay)),STR2:='.csv');
	DirRawdata:= CONCAT(STR1 := CONCAT(STR1 := CONCAT(STR1 := CONCAT(STR1 := CONCAT(STR1 := CONCAT(STR1 := CONCAT(STR1 := CONCAT(STR1 := CONCAT(STR1 := Concat(STR1 := Concat(STR1 := IN_Directory, STR2 := WORD_TO_STRING(TimeStructYesterday.wYear)), STR2 := '\'), STR2 := WORD_TO_STRING(TimeStructYesterday.wMonth)), STR2 := '\'), STR2:='RAWDATA_'), STR2:= WORD_TO_STRING(TimeStructYesterday.wYear)), STR2:='-'),STR2:=WORD_TO_STRING(TimeStructYesterday.wMonth)),STR2:='-'),STR2:=WORD_TO_STRING(TimeStructYesterday.wDay)),STR2:='.csv');
	StartProcess
	(
		NETID := '',
		PATHSTR := 'C:\Windows\System32\compact.exe',
		DIRNAME := 'C:\Windows\System32',
		COMNDLINE :=  CONCAT(STR1:=CONCAT(STR1:=CONCAT(STR1:=CONCAT(STR1:=' /c "',STR2:=DirAlarms), str2:='"  "'), STR2:=DirRawdata),str2:='"'),
		Start := RsJour.Q1,
		TMOUT := T#3M
	);
	IF NOT StartProcess.BUSY THEN
		IF NOT StartProcess.ERR THEN
			StartProcess(Start := FALSE);
			RsJour(RESET1:= TRUE);
			RsJour(RESET1:= FALSE);
		ELSE
			StartProcess(Start := FALSE);
		END_IF
	END_IF	
END_IF

END_FUNCTION_BLOCK

// ---- 00_FunctionsBlocks/Common/DataProcessing/FB_Average.TcPOU
FUNCTION_BLOCK  FB_Average
//////////////////
// Calculate the (fixed) Average of a data ( finishing convention )
//////////////////
VAR_INPUT
	ValueIn 			: ANY ; // Value to average
	WindowDuration		: LINT ; // (ms) Window of Time during which the average will be done 
	CycleTime			: INT := CstCycleTime_G; // (ms) Cycle time of the CPU
END_VAR
	
VAR_OUTPUT
	ValueOut			: REAL ; // Averaged Value. 
	bError 				: BOOL ; // Switch to true if error i inputs				
END_VAR

VAR
	ValueSum			: REAL ; 							// intermediate Sum value of data in fixed Window range. 
	pAnyReal			: POINTER TO REAL;
	pAnyLReal			: POINTER TO LREAL;
	pAnyULint			: POINTER TO ULINT;
	pAnyUint			: POINTER TO UINT;
	NbPoints			: LINT ; 	// Number of points used for calculating the average. 
	
	JJ					: DINT;		// Pick Up index .
	
END_VAR

// EVALUATE VARIABLES //
NbPoints 		:= WindowDuration 	/ 	CycleTime  ;  // Number of Cycle in the Window
//Ceci est un test pour la subversion. KBT
// CHECK INPUTS //
IF NbPoints =0 THEN 
	bError 		:= TRUE ; 
	ValueOut 	:= -1 ;
	
ELSE
	IF (ValueIn.TypeClass = __SYSTEM.TYPE_CLASS.TYPE_REAL) THEN
		pAnyReal        := ValueIn.pValue; 
		ValueSum  		:= ValueSum + (pAnyReal^);
	ELSIF (ValueIn.TypeClass = __SYSTEM.TYPE_CLASS.TYPE_LREAL) THEN
		pAnyLReal     	:= ValueIn.pValue; 
		ValueSum  		:= ValueSum +  LREAL_TO_REAL(pAnyLReal^);
	ELSIF (ValueIn.TypeClass = __SYSTEM.TYPE_CLASS.TYPE_ULINT) THEN
		pAnyULint     	:= ValueIn.pValue; 
		ValueSum  		:= ValueSum +  ULINT_TO_REAL(pAnyULint^);
	ELSIF (ValueIn.TypeClass = __SYSTEM.TYPE_CLASS.TYPe_uint) THEN
		pAnyUint		:= ValueIn.pValue;
		ValueSum		:= ValueSum + UINT_TO_REAL(pAnyUint^);
	END_IF
	JJ			:=JJ+1 ;
	
	IF JJ >= NbPoints THEN  // in order to reset if online change of Cycle time
		ValueOut 	:= ValueSum / LINT_TO_REAL(NbPoints)  ; // Average
		ValueSum 	:= 0 ; 	// Reinitialize sum
		JJ			:= 0 ; // Reinitialize JJ

	END_IF

END_IF

END_FUNCTION_BLOCK

// ---- 00_FunctionsBlocks/Beckhoff/Annexesfunction/FB_RestartService.TcPOU
FUNCTION_BLOCK FB_RestartService
VAR_INPUT
	IN_Directory			: T_MaxString; // directory of the file to compress
	ParamNetID				: STRING ; // Net ID of the PC with HH collector
	IN_ServiceName			: STRING  ;
	Start					: BOOL;
END_VAR
VAR
	StartProcess 			: NT_StartProcess;
	TrigStart				: R_TRIG;
END_VAR

TrigStart(CLK:=Start);
	StartProcess
	(
		NETID := ParamNetID,
		PATHSTR := concat(str1:= IN_Directory, str2 := IN_ServiceName),
		DIRNAME := IN_Directory,
		COMNDLINE := '',
		Start := TrigStart.Q,
		TMOUT := T#3M
	);
	IF NOT StartProcess.BUSY THEN
		IF NOT StartProcess.ERR THEN
			StartProcess(Start := FALSE);
		ELSE
			StartProcess(Start := FALSE);
		END_IF
	END_IF

END_FUNCTION_BLOCK

// ---- 00_FunctionsBlocks/Beckhoff/Annexesfunction/FUN_GetPublicIp.TcPOU
PROGRAM FUN_GetPublicIp

VAR_INPUT
	ParamNetID				: STRING :='' ; // Unit ID of the PC with internet connexion
	IN_CmdStart 			: BOOL;
	IN_DirExe				: STRING;
END_VAR
VAR_OUTPUT
	OUT_Completed			: BOOL;
END_VAR

VAR
	RS_Start				: RS;
	TRIG_Completed			: R_TRIG;
	TRIG_Start				: R_TRIG;
	start_process			: NT_StartProcess;
END_VAR


TRIG_Start(ClK := IN_CmdStart);
TRIG_Completed(CLK := OUT_Completed);


RS_Start(SET := TRIG_Start.Q, RESET1 := TRIG_Completed.Q);

IF RS_Start.Q1 THEN
	IN_CmdStart := FALSE;
	start_process
	(
		NETID := ParamNetID,
		PATHSTR := Concat(IN_DirExe, 'GetPublicIp.exe'),
		DIRNAME := IN_DirExe,
		COMNDLINE := '',
		Start := TRUE
	);
ELSE
	start_process(START := FALSE);
END_IF

IF TRIG_Completed.Q THEN
	OUT_Completed := FALSE;
END_IF

END_PROGRAM

// ---- 00_FunctionsBlocks/Beckhoff/Annexesfunction/FUN_ConnectVPN.TcPOU
PROGRAM FUN_ConnectVPN

VAR_INPUT
	ParamNetID				: STRING :='' ; // Unit ID of the PC with internet connexion
	IN_CmdStart 			: BOOL;
	IN_DirExe				: STRING;
	IN_OpenVpnFile			: STRING;
END_VAR
VAR_OUTPUT
	OUT_Completed			: BOOL;
END_VAR

VAR
	RS_Start				: RS;
	TRIG_Completed			: R_TRIG;
	TRIG_Start				: R_TRIG;
	start_process			: NT_StartProcess;
	TRIG_Available			: F_TRIG;
	bTest: BOOL;
END_VAR


TRIG_Start(CLK := IN_CmdStart);

start_process
(
	NETID := ParamNetID,
	PATHSTR := '"C:\Program Files\OpenVPN\bin\openvpn-gui.exe"',
	DIRNAME := 'C:\Program Files\OpenVPN\bin',
	COMNDLINE := Concat(str1 := '--command connect ', str2 := concat(STR1 := IN_OpenVpnFile, STR2 := '.ovpn')),
	Start := TRIG_Start.Q
);

END_PROGRAM

// ---- 00_FunctionsBlocks/Beckhoff/Annexesfunction/FUN_DisconnectVPN.TcPOU
PROGRAM FUN_DisconnectVPN

VAR_INPUT
	ParamNetID				: STRING :='' ; // Unit ID of the PC with internet connexion
	IN_CmdStart 			: BOOL;
	IN_DirExe				: STRING;
END_VAR
VAR_OUTPUT
	OUT_Completed			: BOOL;
END_VAR

VAR
	TRIG_Start				: R_TRIG;
	start_process			: NT_StartProcess;
END_VAR

TRIG_Start(ClK := IN_CmdStart);

start_process
(
	NETID := ParamNetID,
	PATHSTR := '"c:\Program Files\OpenVPN\bin\openvpn-gui.exe" ',
	DIRNAME := 'C:\Program Files\OpenVPN\bin',
	COMNDLINE := '--command disconnect_all',
	Start := TRIG_Start.Q
);

END_PROGRAM

// ---- 00_FunctionsBlocks/Beckhoff/Annexesfunction/PRG_RestartPlc.TcPOU
PROGRAM PRG_RestartPlc
VAR
END_VAR
VAR_INPUT
	CmdRestart 	: BOOL;
END_VAR

VAR
	RestartProcess : NT_Reboot;
	Trig_Restart	: R_TRIG;
	
END_VAR

Trig_Restart(CLK := CmdRestart);

RestartProcess
(
	NETID := '',
	START := Trig_Restart.Q,
	DELAY := 5,
	TMOUT := T#1S
);

END_PROGRAM

// ---- 04_Application/COM/ModbusTcp.TcPOU
PROGRAM ModbusTcp
Var
    MW  : FB_SplitRealToWords_IEEE754;
    MW1  : FB_SplitUlintToWords;
(*
   mySimpleTcpServer: FbMbSimpleServerTcp :=(  xOpen           := TRUE,  wPort := 2000,bUnitId := 1,
                                              utKeepAlive     := (xEnable      := TRUE, //  Switch keep-alive mechanism on
                                                                       tMaxIdleTime := T#5S, //  Maximum time of inactivity
                                                                        tInterval    := T#2S, //  Interval between two successive KA-Packets
                                                                     udiProbes    := 5 ));    //  Number of KA retry before giving up
*)
END_VAR


(* 
//--- Call the server --------------------------------------------- 
mySimpleTcpServer(  awHoldingRegisters  := GVL_DataBaseStructures.AX_StructModbusTCP    ); 
 *)

END_PROGRAM

// ---- 00_FunctionsBlocks/Common/DataProcessing/SplitWord/FB_SplitRealToWords_IEEE754.TcPOU
FUNCTION_BLOCK FB_SplitRealToWords_IEEE754
VAR_INPUT
	IN_Real : REAL;
END_VAR
VAR_OUTPUT
	OUT_WordStrong :  WORD;
	OUT_WordWeak :  WORD;

END_VAR
VAR

END_VAR

MEMCPY(destAddr := ADR(OUT_WordStrong), srcAddr := ADR(IN_Real), n := 2);
MEMCPY(destAddr := ADR(OUT_WordWeak), srcAddr := ADR(IN_Real) + 2, n := 2);

END_FUNCTION_BLOCK

// ---- 00_FunctionsBlocks/Common/DataProcessing/SplitWord/FB_SplitUlintToWords.TcPOU
FUNCTION_BLOCK FB_SplitUlintToWords
VAR_INPUT
	IN_ULINT : ULINT;
END_VAR
VAR_OUTPUT
	OUT_WorDS_Transfoong :  WORD;
	OUT_WordWeak :  WORD;

END_VAR
VAR

END_VAR

MEMCPY(destAddr := ADR(OUT_WorDS_Transfoong), srcAddr := ADR(IN_ULINT), n := 2);
MEMCPY(destAddr := ADR(OUT_WordWeak), srcAddr := ADR(IN_ULINT) + 2, n := 2);

END_FUNCTION_BLOCK

// ---- 00_FunctionsBlocks/Beckhoff/AlarmManagement/FUN_ReadAlarm_CSV.TcPOU
PROGRAM FUN_ReadAlarm_CSV
//Permet de lire les Valeurs de max 1 semaine de points (1 pt/min pdt 7 jours)

VAR_INPUT
	InDirectory_Stockage 		: T_MaxString;		// Base file of the Historization 
	InStartTimeStamp			: TIMESTRUCT;
	InExecute					: BOOL;			//Rising Edge detection of read
	ParamSeparateur				: STRING;
	IN_Reset					: BOOL ; // Close File . 
	ParamMaxLine				: WORD :=  200 ; 
END_VAR                 		

VAR_OUTPUT              		
	OutValue					: ARRAY[1..500] OF ST_ValuesAlarms;
	OutDir						: T_Maxstring;
	OutCompleted				: BOOL;
	OutNbLigne					: UINT;
	OutbBusy					: BOOL;
	OutError 					: BOOL;
	OutErrorID 					: UINT; // 1 : File not found
END_VAR                 		
VAR     
	// Initialisation 
	TypeFile					: STRING;
	ParamTimeOut				: TIME := T#1S;
	
	//Read
	TimeStructBeingRead			: TIMESTRUCT;
	FullDirectory				: STRING;                		
	
	OpenFile					: FB_FileOpen;
	ReadFile					: FB_FileGets;
	CloseFile					: FB_FileClose;
	InfoFile					: FB_EnumFindFileEntry;
	FileInfo					: ST_FindFileEntry;

	Index_Array_OutValue		: UINT := 1;			// Valeur de OutValue qui va être écrite
	
	Opening						: BOOL := TRUE;
	
	LineRead					: T_Maxstring;
	EOF_Reached					: BOOL;              		
	CompteurLigne				: CTU;
	AX_ArrayString 				: ARRAY[1..100] OF T_Maxstring;
	
	OutEmpty					: ARRAY[1..500] OF ST_ValuesAlarms;
	OutBusy						: RS;
	OutCompleted_RS				: RS;
	Trig_Read					: R_TRIG;
	Trig_Start 					: R_TRIG;
	
	FileHandle					: UINT;
	FileHandle_Old				: UINT;
	
	KK: UINT := 1;
	bInit : BOOL;
	LL: UINT;
	MM: UINT;
END_VAR

Trig_Start(CLK := InExecute);
OutCompleted_RS(Reset1 := Trig_Start.Q);
IF trig_start.Q THEN
	OutEmpty := OutValue;
	outError := FALSE;
END_IF
OutBusy(Set := InExecute, RESET1 := OutError OR OutCompleted_RS.Q1);
OutbBusy := OutBusy.Q1;
OutCompleted := OutCompleted_RS.Q1;
IF OutBusy.Q1 THEN	
	// J'initialise le tout : 
	//Initialisation du type de fichier
	TypeFile := 'ALARMS'; 
	
	TimeStructBeingRead := DT_TO_SYSTEMTIME(SYSTEMTIME_TO_DT(InStartTimeStamp) );
	FullDirectory := Concat(Concat(Concat(Concat(Concat(Concat(Concat(Concat(Concat(Concat(Concat(Concat(InDirectory_Stockage , WORD_TO_STRING(TimeStructBeingRead.wyear)),'\'),WORD_TO_STRING(TimeStructBeingRead.wMonth)),'\'),'ALARMS'),'_'),WORD_TO_STRING(TimeStructBeingRead.wyear)),'-'),WORD_TO_STRING(TimeStructBeingRead.wMonth)),'-'),WORD_TO_STRING(TimeStructBeingRead.wDay)),'.csv');
    OutDir := FullDirectory;
	//Ouverture du Fichier, récupération du handle
	OpenFile
	(
		sNetId := '',
		sPathName := FullDirectory,
		nMode := FOPEN_MODEREAD,
		ePath := PATH_GENERIC,
		bExecute := Opening AND NOT OutCompleted_RS.Q1,
		hFile => FileHandle
	);
	
	IF OpenFile.nErrId = 1804 THEN // Le fichier n'existe pas 
		OutErrorID := 1;
		OutError := OpenFile.bError;
		OpenFile(bExecute :=  FALSE);
	ELSIF OpenFile.bError THEN		// Il y a eu une autre erreur
		OutError := OpenFile.bError;
	ELSIF NOT OpenFile.bError AND NOT OpenFile.bBusy AND FileHandle <> 0 AND FileHandle <> FileHandle_Old THEN
		opening := FALSE;
		FileHandle_Old := FileHandle;
	END_IF
	// On a obtenu le file handle, on va commencer la lecture

	// Le bloc suivant va lire le document ligne à ligne en incrémentant le compteur ligne et en ressortant l'ensemble de la ligne dans LineRead
	LineRead := '';
	IF NOT opening THEN
		ReadFile
		(
			sNetId := '',
			hFile := FileHandle,
			bExecute := TRUE,
			tTimeout := ParamTimeOut,
			sLine => LineRead,
			bEOF => EOF_Reached
		);				

		IF NOT ReadFile.bBusy AND NOT ReadFile.bError AND (LineRead <> '') THEN
			ReadFile(bExecute := FALSE);
			CompteurLigne(CU := TRUE);	
			CompteurLigne(CU := FALSE);
			IF CompteurLigne.CV > 2 THEN
				Split(IN_TextToSearch := LineRead, IN_Delimiter := 	ParamSeparateur, OUT_Split => AX_ArrayString);			
				OutValue[Index_Array_OutValue].TimeStamp_Act 	:= AX_ArrayString[1];
				OutValue[Index_Array_OutValue].ID 				:= STRING_TO_UINT(AX_ArrayString[2]);
				OutValue[Index_Array_OutValue].Message			:= AX_ArrayString[3];
				OutValue[Index_Array_OutValue].Value			:= STRING_TO_BOOL(AX_ArrayString[4]);
				OutValue[Index_Array_OutValue].Ack			 	:= STRING_TO_BOOL(AX_ArrayString[5]);
				OutValue[Index_Array_OutValue].Alarms_LVL	 	:= STRING_TO_UINT(AX_ArrayString[6]);				
				Index_Array_OutValue := Index_Array_OutValue + 1;
				
			END_IF
		
		ELSIF NOT ReadFile.bBusy AND  ReadFile.bError THEN
			OutError := TRUE;	
		ELSIF  EOF_Reached THEN
			OutNbLigne := Index_Array_OutValue;
			OutCompleted_RS( SET := TRUE);
			OutCompleted_RS( SET := FALSE);
	
		END_IF	
	
	END_IF
	
ELSIF EOF_Reached AND FileHandle <> 0 THEN
	ReadFile(bExecute := FALSE);
	CloseFile
	(
		sNetId := '',
		bExecute := TRUE,
		hFile := FileHandle,
		tTimeout := ParamTimeOut
	);
	IF NOT CloseFile.bBusy AND NOT CloseFile.bError THEN
		CloseFile(bExecute := FALSE);
		Opening := TRUE;
		CompteurLigne(RESET := TRUE);
		CompteurLigne(RESET := FALSE);
		Index_Array_OutValue := 1;
		FileHandle := 0;
		OutValue := OutEmpty;
	ELSIF NOT CloseFile.bBusy AND closefile.bError THEN
		OutError := TRUE;
	END_IF  
END_IF

END_PROGRAM

// ---- 00_FunctionsBlocks/Beckhoff/Annexesfunction/FUN_PingHost.TcPOU
PROGRAM FUN_PingHost
VAR_INPUT
	IN_bStart			: BOOL;	
	IN_PingAdr			: STRING(50);
	IN_DirBatLocation	: STRING(255);
END_VAR
VAR_OUTPUT
	OUT_Result			: BOOL;
	OUT_Completed 		: BOOL;
	OUT_Busy			: BOOL;
	OUT_Error			: BOOL;
END_VAR
VAR
	ReadLine			: T_MaxString;
	ReadResult 			: T_MAXString;
	StartProcess 		: NT_StartProcess;
	TP_StartFunction	: TP;
	TP_StartProcess		: TP;
	RS_Start			: RS;
	Trig_Start			: R_TRIG;
	FB_Read 			: FB_READ;
	Outvalue			: STRING(255);
END_VAR

Trig_Start(CLK := IN_bStart);
IF Trig_Start.Q THEN 
	ReadResult := '';
END_IF
RS_Start(Set := Trig_Start.Q, RESET1 := OUT_Completed);
OUT_Busy := FALSE;
OUT_Completed := FALSE;

IF RS_Start.Q1 THEN
	//Phase de start du processus
	OUT_Busy := TRUE;
	TP_StartProcess(IN := RS_Start.Q1, PT := T#7S);
	StartProcess
	(
		NETID := '',
		PATHSTR:= CONCAT(IN_DirBatLocation, 'PingHost.bat'),
		DIRNAME := IN_DirBatLocation,
		COMNDLINE := IN_PingAdr,
		Start := RS_Start.Q1,
		TMOUT := T#7S
	);
	
	//Phase d'analyse du processus
	IF NOT StartProcess.BUSY AND NOT StartProcess.ERR  AND NOT TP_StartProcess.Q THEN
		FB_Read
		(
			InDirectory := CONCAT(IN_DirBatLocation, 'Ping.txt'),
			InExecute := TRUE,
			OutValue => ReadLine
		);
		
		IF NOT FB_Read.OutbBusy AND NOT fb_read.OutError THEN
			OUT_Completed := TRUE;
			OUT_Busy := FALSE;
			TP_StartProcess(in := FALSE);
			FB_Read(InExecute := FALSE);
			StartProcess(Start := FALSE);
			
			IF left(ReadLine, 14) = 'host reachable' THEN
				ReadResult := 'PING OK';
				OUT_Result := TRUE;
			ELSE
				OUT_Result := FALSE;
				ReadResult := 'PING NOT OK';

			END_IF
		END_IF
	ELSIF NOT StartProcess.BUSY AND StartProcess.ERR THEN
		Out_Error := TRUE;
	END_IF
END_IF

END_PROGRAM

// ---- 00_FunctionsBlocks/Beckhoff/DataProcessing/ReadFile/FB_Read.TcPOU
FUNCTION_BLOCK FB_Read
//Permet de lire les Valeurs de max 1 semaine de points (1 pt/min pdt 7 jours)

VAR_INPUT
	InDirectory 				: T_MaxString;		// Base file of the Historization 
	InExecute					: BOOL;			//Rising Edge detection of read
END_VAR                 		

VAR_OUTPUT              		
	OutValue					: T_MaxString;
	OutCompleted				: BOOL;
	OutbBusy					: BOOL;
	OutError 					: BOOL;
	OutErrorID 					: UINT; // 1 : File not found

END_VAR                 		
VAR     
	// Initialisation 
	RS_Busy						: RS;
	Trig_Start 					: R_TRIG;
	FullDirectory				: STRING;  
	
	OpenFile					: FB_FileOpen;
	ReadFile					: FB_FileRead;
	CloseFile					: FB_FileClose;
	
	Opening						: BOOL := TRUE;
	Reading						: BOOL;
	Closing						: BOOL;
	
	EOF_Reached					: BOOL;
	
	FileHandle					: UINT;
	FileHandle_Old				: UINT;
	
	NbJours						: UINT;
	KK: UINT 					:= 1;
END_VAR

Trig_Start(CLK := InExecute);

IF Trig_Start.Q THEN 
	Outerror:= FALSE ; // On reinitialize l'error à un nouvel essai . 
	OpenFile(bExecute:= FALSE  ); 
END_IF

RS_Busy(Set := Trig_Start.Q, RESET1 := Outerror OR OutCompleted);
OutbBusy := RS_Busy.Q1;
OutCompleted := FALSE;


IF RS_Busy.Q1 THEN	
		//Ouverture du Fichier, récupération du handle
		OpenFile
		(
			sNetId := '',
			sPathName := InDirectory,
			nMode := FOPEN_MODEREAD,
			ePath := PATH_GENERIC,
			bExecute := TRUE,
			hFile => FileHandle
		);
		
		IF NOT OpenFile.bBusy AND OpenFile.bError AND OpenFile.nErrId = 1804 THEN // Le fichier n'existe pas 
			OutErrorID := 1;
			OutError := OpenFile.bError;
		ELSIF OpenFile.bError THEN		// Il y a eu une autre erreur
			OutError := OpenFile.bError;
		ELSIF NOT OpenFile.bError AND NOT OpenFile.bBusy AND FileHandle <> 0 THEN
			opening := FALSE;
		END_IF
		
		
		
		IF NOT opening AND NOT EOF_Reached THEN			
			ReadFile
			(
				sNetId := '',
				hFile := FileHandle,
				bExecute := TRUE,
				tTimeout := T#1S,
				pReadBuff := ADR(OutValue),
				cbReadLen := SIZEOF(OutValue),				
				bEOF => EOF_Reached
			);	
			IF NOT ReadFile.bBusy AND ReadFile.bError THEN
				OutError := TRUE;	
				ReadFile(bExecute := FALSE);
			ELSIF NOT ReadFile.bBusy THEN
				ReadFile(bExecute := FALSE);	
			END_IF
		ELSIF EOF_Reached THEN
			ReadFile(bExecute := FALSE);
	
			CloseFile
			(
				sNetId := '',
				bExecute := TRUE,
				hFile := FileHandle,
				tTimeout := T#1S
			);
			IF NOT CloseFile.bBusy AND NOT CloseFile.bError  THEN
				Opening := TRUE;
				EOF_Reached := FALSE;
				OpenFile(bExecute := FALSE);
				ReadFile(bExecute := FALSE);
				CloseFile(bExecute := FALSE);
				
				OUTCompleted := TRUE;
			ELSIF CloseFile.bError THEN
				OutError := TRUE;
				OutErrorID := UDINT_TO_UINT(Closefile.nErrId);
			END_IF	
		END_IF
	END_IF

END_FUNCTION_BLOCK

// ---- 00_FunctionsBlocks/Beckhoff/Communication/IEC104/FB_IEC104ServerAkuo.TcPOU
FUNCTION_BLOCK FB_IEC104ServerAkuo
VAR_INPUT
	protPara  		: ST_IEC870_5_104ProtocolParams ;	// protocol parameters 
	sysPara	  		: ST_IEC870_5_101SystemParams ; 	// system parameters. 
	akuoPara		: ST_IEC104AkuoParam;				// akuo parameters. 
	
	IN_bEnable		: BOOL := TRUE ;					// enable or disable IEC 104 Server  .
	IN_Local		: BOOL ;  							// Server in local. Data flow is inhibated in control direction, allow in monitor direction.  
	IN_CmdReset		: BOOL ;							// Reset after a change in the protPara , or  sysPara
	
	memory 			: PVOID ; 							// ADR() . Pointer to starting address. 	
	AODB 			: ARRAY[0..GVL_Cst.CstNbAOEntries] OF ST_IEC870_5_101AODBEntry ;	// AODB	
END_VAR

VAR_OUTPUT
	eConnState		: E_SocketConnectionState := eSOCKET_DISCONNECTED;
	eDTState		: E_IEC870_5_104DataTransferState := eIEC870_STOPDT ;
END_VAR
VAR
// M_INIT 
	bInit					: BOOL := TRUE;

//M_PREPAREAO // 
	nBytesRead				: ARRAY[0..GVL_Cst.CstNbAOEntries] OF UDINT;		// Number of bytes taken by the raw data ( float = 4  SIQ = 1 , ...)
	Mask					: ARRAY[0..GVL_Cst.CstNbAOEntries] OF  DWORD;		// Mask corresponding to number of byte above . 
	MesCmd_old				: ARRAY[0..GVL_Cst.CstNbAOEntries] OF DWORD ; 		// Value in the memory space ( after bytes and bit offset ). 
	MesDword_Old			: ARRAY[0..GVL_Cst.CstNbAOEntries] OF DWORD;		// Raw dword value in memory space . 
	FB_Flicker				: ARRAY[0..GVL_Cst.CstNbAOEntries] OF FB_DetectFlicker ; 	// Function to detect flickering 

// M_CONNECT //
	hServer					: T_HSERVER; // TCP/IP server handle
	eComState				: E_ComState	:= INIT;
	fbConnection			: FB_ServerClientConnection;
	fbProtocol				: FB_IEC870_5_104TProtocol;

// TIME MANAGEMEMENT //
	systemTime_CP56Time2a			: T_CP56Time2a;
	FB_LocalSystTime				: FB_LocalSystemTime;
	CalLocalTimeStruct				: TIMESTRUCT ; 
	
// PROCESS DATA 
	stBuffer				: ST_IEC870_5_101TBuffer;		// Buffer of data to send in monitoring direction
	fbBuffer				: FB_IEC870_5_101TBufferCtrl;	// Buffer of data to send in control direction . 
	
	stTxAsdu 				: ST_IEC870_5_101AOGen; 	// asdu to be send . Copied from current AO . 
	KK						: INT ;	// loop 
	JJ						: INT;	// loop
	
// M_READCMD //
	stRxAsdu 				: ST_IEC870_5_101AOGen; // received asdu 
	nQOI					: BYTE;		// general interrogation data
	fbsetLocalTime			: NT_SetLocalTime; //clock synchronisation time apply

// M_CYCLIC // 
	fbCyclicTime				: TON;	// Cyclic trigger

//M_CHANGE DATA//
	CmdOldValue				: ARRAY[0..GVL_Cst.CstNbAOEntries] OF DWORD;		// Value of predecessing commAND  

END_VAR

IF bInit OR IN_CmdReset THEN 
	M_Init() ;
	bInit := FALSE ; 
END_IF

M_PrepareAO(); 

// GET LOCAL TIME AND CONVERT TO CP56Time 
FB_LocalSystTime(
	bEnable := TRUE,
	dwCycle := 1,
	systemTime => CalLocalTimeStruct);
		 
systemTime_CP56Time2a := SYSTEMTIME_TO_CP56Time2a(TIMESTR := CalLocalTimeStruct, SU := FALSE);

// Connexion management 
M_Connect();

// Read Command in control direction//
M_ReadCmd() ;

// Cyclic Data in monitoring direction//
fbCyclicTime(IN:= sysPara.bPerCyclic XOR fbCyclicTime.Q, PT:= sysPara.tPerCyclicBase);
IF sysPara.bPerCyclic AND fbCyclicTime.Q AND (eComState = DATATRANSFER) THEN
	M_Cyclic();
END_IF

// On change data in monitoring direction//
IF (eComState = DATATRANSFER) THEN
	M_ChangeData();
END_IF

METHOD M_ChangeData : BOOL
VAR_INPUT
END_VAR
FOR KK := 0 TO akuoPara.iAOnb DO 
	IF AODB[KK].aObj.obj.ident.eType = 30 OR AODB[KK].aObj.obj.ident.eType = 31 THEN 
		// Get value of corresponding byte .
		IF CmdOldValue[KK]<> MesCmd_old[KK] THEN 
			CmdOldValue[KK] := MesCmd_old[KK] ;
			stTxAsdu :=  AODB[KK].aObj.obj ; 
			stTxAsdu.ident.eCOT		:= eIEC870_COT_SPONTAN;	// cause of transmission - spontaneous
			stTxAsdu.ident.nORG		:= sysPara.orgAddr;				// originator address

			fbBuffer.TxAddObj(putObj := stTxAsdu,buffer := stBuffer);
			IF NOT fbBuffer.bOk THEN
				// code for buffer overflow
				RETURN; 
			END_IF	 		
		END_IF
	END_IF
END_FOR
END_METHOD

METHOD M_Connect : BOOL
VAR_INPUT
END_VAR

VAR

END_VAR
// connection management
CASE eComState OF
INIT: 
	// INIT protocol parameter
	fbConnection.eMode		:= eACCEPT_ALL;	// accept all incomming connections
	fbConnection.tReconnect	:= T#2S;
	
	fbProtocol.sSrvNetID				:= '';		
	fbProtocol.protPara.bPackFrames		:= TRUE;
	fbProtocol.protPara.bThrottleMode	:= protPara.bThrottleMode;
	fbProtocol.bOutDbg					:= FALSE;	// disable debug output


	// INIT RX/TX buffer parameter
	stBuffer.eDbg					:= eIEC870_FIFO_DBG_ALL;
	stBuffer.asduFmt.eCOTSize		:= eIEC870_COT_TwoOctets;		// cause of transfer size
	stBuffer.asduFmt.eAsduAddrSize	:= eIEC870_AsduAddr_TwoOctets;	// common asdu addr size
	stBuffer.asduFmt.eObjAddrSize	:= eIEc870_ObjAddr_ThreeOctets;	// object address size

	eComState := IDLE;
	
	
IDLE:	
	IF IN_bEnable THEN
		F_CreateServerHnd(	bEnable		:= FALSE,
							sSrvNetID	:= '',			// own (server) NetID
							sLocalHost	:= akuoPara.sLocalHost ,
							
							nLocalPort	:= akuoPara.iLocalPort,
							nMode		:= LISTEN_MODE_CLOSeALL OR CONNECT_MODE_ENABLEDBG, // Close all previous opened and not closed sockets and enable debug messages on socket creation/connect/close
							hServer		:= hServer );	// create server connection handle
						
		stBuffer.asduSize := F_iecApdu104ToAsduLen(fbProtocol.protPara.APDULength);
		eComState := CONNECT;
	END_IF

	
CONNECT: 
	fbConnection( 	bEnable := IN_bEnable,
					hServer	:= hServer );		
			
	CASE fbConnection.eState OF 
		eSOCKET_CONNECTED:
		
			fbProtocol.INIT( 	hSocket	:= fbConnection.hSocket, // reset fbProtocol and restart data transfer
								buffer	:= stBuffer );
			eComState := DATATRANSFER;			
		eSOCKET_DISCONNECTED:
			eComState := IDLE;	
		eSOCKET_SUSPENDED:
			; // wait for connection	
	END_CASE		
		eConnState := fbConnection.eState ;

DATATRANSFER: 
	IF IN_bEnable THEN
		fbProtocol(buffer := stBuffer);
		 eDTState := fbProtocol.eDTState ;
		IF NOT fbProtocol.bError THEN
			IF fbProtocol.eDTState = eIEC870_STARTDT THEN	
				;// exchange data
			END_IF
		ELSE // error occured - log error msg. and close socket
			(*ADSLOGSTR(	ADSLOG_MSGTYPE_ERROR OR ADSLOG_MSGTYPE_LOG,		// log errors
						'IEC60870-5-104 Transport Interface error: %s',
						DWORD_TO_HEXSTR(fbProtocol.nErrID,0,TRUE)); *)
			eComState := DISCONNECT;
		END_IF
	ELSE // stop data transfer
		eComState := DISCONNECT;
	END_IF

	
DISCONNECT: 
	fbProtocol(buffer := stBuffer);	
	fbConnection(	hServer := hServer,
					bEnable := FALSE );
					
	IF fbConnection.eState = eSOCKET_DISCONNECTED 
	AND fbProtocol.eDTState = eIEC870_STOPDT THEN
		eComState := IDLE;
	END_IF
END_CASE
END_METHOD

METHOD M_Cyclic : BOOL
VAR_INPUT
END_VAR
// Data, cyclic	
//##############################################################################################################################################//	

FOR KK := 0 TO akuoPara.iAOnb DO 
	IF AODB[KK].aObj.cfg.group.30 AND AODB[KK].aObj.obj.ident.eType<>0 THEN 
		stTxAsdu :=  AODB[KK].aObj.obj ; 

		stTxAsdu.ident.eCOT		:= eIEC870_COT_CYCLIC;	// cause of transmission - spontaneous
		stTxAsdu.ident.nORG		:= sysPara.orgAddr;				// originator address
		fbBuffer.TxAddObj(	putObj := stTxAsdu,buffer := stBuffer);
		IF NOT fbBuffer.bOk THEN
			// code for buffer overflow
			RETURN; 
		END_IF
	END_IF
END_FOR
END_METHOD

METHOD M_Init : BOOL
VAR_INPUT
END_VAR

VAR

END_VAR
END_METHOD

METHOD M_PrepareAO : BOOL
VAR_INPUT
END_VAR
VAR
	bAddCPTime		: BOOL;		// IF CP56Time is attached
	bAddQDS			: BOOL;		// If QDS is in a separate BYTE 
	QDS				: BYTE;		// QDS Value ( Quality descriptor )
	IV				: BOOL;		// INvalid
	SB				: BOOL;		//
	NT				: BOOL;		// Not topical
	BL				: BOOL;		// Blocked

	bFlicker		: BOOL;		// detect if data is flickering 

END_VAR
FOR KK := 0 TO akuoPara.iAOnb DO 
	AODB[KK].aObj.obj.ident.asduAddr	:= sysPara.asduAddr;
	AODB[KK].aObj.obj.ident.eClass		:= eIEC870_Class_1;
	
	// Get value in memory space. 
	F_iecResetStream(0,AODB[KK].aObj.obj.info.stream);
	MEMCPY( destAddr := ADR(MesDword_Old[KK]) , srcAddr := memory+ULINT_TO_DWORD(AODB[KK].aObj.cfg.byteOffs) , n := nBytesRead[KK]);
	MesCmd_old[KK] := SHR(MesDword_Old[KK] , AODB[KK].aObj.cfg.bitOffs) AND Mask[KK] ;

	CASE AODB[KK].aObj.obj.ident.eType OF 
		30:	// 
			AODB[KK].aObj.obj.ident.nObj		:= 1;
			nBytesRead[KK] := 1 ; 
			Mask[KK] := 2#1 ;
			bAddCPTime := TRUE ;
			bAddQDS		:= FALSE ;

			FB_Flicker[KK](IN_VAR:= MesCmd_old[KK].0	, IN_Window := akuoPara.tFlickerWindow , IN_COUNT:= akuoPara.uFlickerNumber , OUT_bFlicker => bFlicker );

			IF bFlicker AND akuoPara.bEnableFlicker THEN 
				BL := TRUE ;
				IV := TRUE ;
				MesCmd_old[KK].0 := 0 ;	// Freeze value .
			ELSE 
				BL := FALSE ;
				IV := FALSE ;
			END_IF
			
			
		31:
			AODB[KK].aObj.obj.ident.nObj		:= 1;
			nBytesRead[KK] := 1 ; 
			Mask[KK] := 2#11;
			bAddCPTime := TRUE ;
			bAddQDS		:= FALSE ;
		36:
			AODB[KK].aObj.obj.ident.nObj		:= 1;
			nBytesRead[KK] := 4 ; 
			Mask[KK] := 16#FFFFFFFF;	
			bAddCPTime := TRUE ;
			bAddQDS		:= TRUE ;
		13:
			AODB[KK].aObj.obj.ident.nObj		:= 1;
			nBytesRead[KK] := 4 ; 
			Mask[KK] := 16#FFFFFFFF;	
			bAddCPTime := FALSE ;
			bAddQDS		:= TRUE ;
		58:
			AODB[KK].aObj.obj.ident.nObj		:= 1;
			nBytesRead[KK] := 1 ; 
			Mask[KK] := 16#1;	
			bAddCPTime := TRUE ;		
			bAddQDS		:= FALSE ;	
	
		59:
			AODB[KK].aObj.obj.ident.nObj		:= 1;
			nBytesRead[KK] := 1 ; 
			Mask[KK] := 2#11;	
			bAddCPTime := TRUE ;
			bAddQDS		:= TRUE ;
			
		63:		// C_SE_TC_1 - Short floating point . 
			AODB[KK].aObj.obj.ident.nObj		:= 1;
			nBytesRead[KK] := 4 ; 
			Mask[KK] := 16#FFFFFFFF;	
			bAddCPTime := FALSE ;	
			bAddQDS		:= TRUE ;		
		
	END_CASE
	
	// Set Quality descriptor
	QDS:= 0;
	QDS.7 :=  IV OR AODB[KK].aObj.sts.bIV_Internal; 
	QDS.6 :=  NT ;
	QDS.5 := SB ; 
	QDS.4 := BL ;
	
	IF 	bAddQDS THEN
		F_iecCopyBufferToStream(ADR(MesCmd_old[KK]),nBytesRead[KK],AODB[KK].aObj.obj.info.stream);	// copy values TO transmit stream
		F_iecCopyBufferToStream(ADR(QDS),SIZEOF(QDS),AODB[KK].aObj.obj.info.stream);	// copy values TO transmit stream
	ELSE	
		MesCmd_old[KK] :=  MesCmd_old[KK] OR QDS ;
		F_iecCopyBufferToStream(ADR(MesCmd_old[KK]),nBytesRead[KK],AODB[KK].aObj.obj.info.stream);	// copy values TO transmit stream
	END_IF

	IF 	bAddCPTime THEN 
		F_iecCopyBufferToStream(ADR(systemTime_CP56Time2a),SIZEOF(systemTime_CP56Time2a),AODB[KK].aObj.obj.info.stream);	// copy values TO transmit stream
	END_IF
END_FOR
END_METHOD

METHOD M_ReadCmd : BOOL
VAR_INPUT
END_VAR
VAR
		MesCmd					: DWORD ;	// Processed command
		TempData_bis			: DWORD ;	// Intermediate variable

		nDCO_Cmd				: BYTE;		// Temporary variable for Double Command
		nSCO_Cmd				: BYTE ;	// Temporary variable for Single Command
		nSCO_Val				: DWORD ;	// Temporary variable for Float Command
		tActTime				: T_CP56Time2a ;
		CountAO 				: BYTE  ;	// detect if wrong IOA received
END_VAR
// -----------------------------------------------------------------------------------
// process received data
REPEAT
	fbBuffer.RxRemoveObj(	getObj => stRxAsdu,
 							buffer := stBuffer);						
	IF fbBuffer.bOk THEN
		CASE stRxAsdu.ident.eType OF
			C_IC_NA_1: 
				// General Interrogation
				F_iecCopyStreamToBuffer (ADR(nQOI),SIZEOF(nQOI), stRxAsdu.info.stream); //Copy value to local varialbe
				// create general interrogation confirmation asdu
				stTxAsdu := stRXAsdu;
				stTxAsdu.ident.eCOT := eIEC870_COT_ACT_CON; // cause of transfer -> activation confirmation
				fbBuffer.TxAddObj(	putObj := stTxAsdu,
									buffer := stBuffer);
				IF NOT fbBuffer.bOk THEN
					// code for buffer overflow (send overflow response) 

					EXIT; 
				END_IF
			
				FOR KK := 0 TO akuoPara.iAOnb DO 
				
					IF AODB[KK].aObj.cfg.group.0 AND AODB[KK].aObj.obj.ident.eType<>0 THEN 
						// create first asdu (bSlaveToMaster)
						AODB[KK].aObj.obj.ident.eCOT		:= BYTE_TO_INT(nQOI);
						AODB[KK].aObj.obj.ident.nORG		:= stRxAsdu.ident.nORG;
						stTxAsdu := AODB[KK].aObj.obj ;
	
						fbBuffer.TxAddObj(	putObj:= stTxAsdu,
											buffer:= stBuffer);
						IF NOT fbBuffer.bOk THEN
							// code for buffer overflow
							EXIT;
						END_IF	
					END_IF				
				END_FOR
				
				// create general interrogation activation termination asdu
				stTxAsdu := stRxAsdu;
				stTxAsdu.ident.eCOT := eIEC870_COT_ACT_TERM;	// cause of transfer -> activation termination
				fbBuffer.TxAddObj(	putObj:= stTxAsdu,
									buffer:= stBuffer);
				IF NOT fbBuffer.bOk THEN
					// code for buffer overflow
					EXIT; 
				END_IF			
			
			C_DC_TA_1:	// Commande Double		26 -> 43 ;	27 ->44
				CountAO := 0 ; 
				FOR KK:=1 TO akuoPara.iAOnb DO 
					IF stRxAsdu.info.objAddr = AODB[KK].aObj.obj.info.objAddr AND stRxAsdu.ident.eType = AODB[KK].aObj.obj.ident.eType THEN 
						CountAO := CountAO +1 ; ;
						F_iecCopyStreamToBuffer(ADR(nDCO_Cmd),SIZEOF(nDCO_Cmd),stRxAsdu.info.stream);
						// Get value of corresponding byte .
						TempData_bis := MesDword_Old[KK] XOR SHL(MesCmd_old[KK] ,AODB[KK].aObj.cfg.bitOffs )  ; 	// We set to zero here the bits that will be replaced
						TempData_bis := SHL(nDCO_Cmd AND Mask[KK] , AODB[KK].aObj.cfg.bitOffs) OR TempData_bis ;	// We insert the new bits 
						
						IF NOT IN_Local	THEN	
							// Apply read only if not in local . 	
							MEMCPY( destAddr := memory+ULINT_TO_DWORD(AODB[KK].aObj.cfg.byteOffs) , srcAddr := ADR(TempData_bis) , n := nBytesRead[KK]);
							MesCmd := nDCO_Cmd AND Mask[KK] ;
						ELSE
							// in local overwrite the command by the former value .
							nDCO_Cmd	:= DWORD_TO_BYTE(MesCmd_old[KK])	;
						END_IF										
						
						IF nDCO_Cmd.7 THEN
							// (1)SELECT / (0) EXECUTE STATE ( not used ) 
							; // code for select bit 
						END_IF
					
						// create activation confirmation asdu
						stTxAsdu := stRxAsdu;
						stTxAsdu.info.stream.data[0] := nDCO_Cmd;	// Permet de mettre à jour que si pas en local
						stTxAsdu.ident.eCOT := eIEC870_COT_ACT_CON; //cause of transfer -> activation confirmation
						IF IN_Local THEN
							stTxAsdu.ident.bPN :=  TRUE;
						ELSE 
							stTxAsdu.ident.bPN := FALSE;
						END_IF	
						
						fbBuffer.TxAddObj(	putObj := stTxAsdu,
											buffer := stBuffer);
						IF NOT fbBuffer.bOk THEN
							// code for buffer overflow
							EXIT; 
						END_IF
						
						IF NOT nDCO_Cmd.7 AND NOT IN_Local THEN	
	
							IF NOT (MesCmd = MesCmd_old[KK] OR IN_Local) THEN
								// Gets corresponding data type.
								stTxAsdu := AODB[KK].aObj.obj ;
								FOR JJ:= 1 TO GVL_Cst.CstNbAOEntries DO 
									IF KK<>JJ AND AODB[KK].aObj.cfg.byteOffs = AODB[JJ].aObj.cfg.byteOffs AND AODB[KK].aObj.cfg.bitOffs = AODB[JJ].aObj.cfg.bitOffs THEN
										stTxAsdu := AODB[jj].aObj.obj ;
										EXIT;
									END_IF
								END_FOR
							
								stTxAsdu.ident.eCOT		:= eIEC870_COT_RETREM;	// cause of transmission - spontaneous
								stTxAsdu.ident.nORG		:= sysPara.orgAddr;				// originator address
								
								F_iecResetStream(0,stTxAsdu.info.stream);
								F_iecCopyBufferToStream(ADR(nDCO_Cmd),SIZEOF(nDCO_Cmd),stTxAsdu.info.stream);	// copy values TO transmit stream
								fbBuffer.TxAddObj(	putObj := stTxAsdu,
													buffer := stBuffer);
								IF NOT fbBuffer.bOk THEN
									// code for buffer overflow
									RETURN; 
								END_IF	
							END_IF					
						END_IF
	
						IF NOT nDCO_Cmd.7 AND NOT IN_Local THEN	
							// code for execute function
							//create command activation termination asdu
							stTxAsdu := stRxAsdu;
							stTxAsdu.ident.eCOT := eIEC870_COT_ACT_TERM; // cause of transfer -> activation termination
							IF MesCmd = MesCmd_old[KK] THEN
								stTxAsdu.ident.bPN :=  TRUE;
							ELSE 
								stTxAsdu.ident.bPN := FALSE;
							END_IF						
					
							fbBuffer.TxAddObj(	putObj := stTxAsdu,
												buffer := stBuffer);
							IF NOT fbBuffer.bOk THEN
								// code for buffer overflow
								EXIT; 
							END_IF				
						END_IF
					END_IF
				END_FOR
				
				IF CountAO = 0 THEN 
					// code for invalid object address	IOA : return command with invalid data . 
						stTxAsdu := stRxAsdu;
						IF stRxAsdu.info.objAddr = AODB[KK].aObj.obj.info.objAddr THEN
							stTxAsdu.ident.eCOT := eIEC870_COT_UNKNOWN_TYPE; // cause of transfer -> Wrong TYPE for this IoA .  
						ELSE
							stTxAsdu.ident.eCOT := eIEC870_COT_UNKNOWN_OBJECT_ADDRESS; // cause of transfer -> unknown IOA 
						END_IF
						
						stTxAsdu.ident.bPN :=  TRUE;					
						fbBuffer.TxAddObj(	putObj := stTxAsdu,
											buffer := stBuffer);
						IF NOT fbBuffer.bOk THEN
							// code for buffer overflow
							EXIT; 
						END_IF				
					EXIT;  
				END_IF
				
			C_SC_TA_1: // single command with time tag 	30-32-33
				CountAO := 0 ; 
				FOR KK:=1 TO akuoPara.iAOnb DO 
					IF stRxAsdu.info.objAddr = AODB[KK].aObj.obj.info.objAddr THEN 
						CountAO := CountAO +1 ; ;
						F_iecCopyStreamToBuffer(ADR(nSCO_Cmd),SIZEOF(nSCO_Cmd),stRxAsdu.info.stream);
						// Get value of corresponding byte .
						TempData_bis := MesDword_Old[KK] XOR SHL(MesCmd_old[KK] ,AODB[KK].aObj.cfg.bitOffs )  ; 	// We set to zero here the bits that will be replaced
						TempData_bis := SHL(nSCO_Cmd AND Mask[KK] , AODB[KK].aObj.cfg.bitOffs) OR TempData_bis ;	// We insert the new bits 
						
						IF NOT IN_Local	THEN				// Permet de mettre à jour la commande que si pas en local
				
							MEMCPY( destAddr := memory+ULINT_TO_DWORD(AODB[KK].aObj.cfg.byteOffs) , srcAddr := ADR(TempData_bis) , n := nBytesRead[KK]);
							MesCmd := nSCO_Cmd AND Mask[KK] ;
						ELSE
							// in local overwrite the command by the former value .
							nSCO_Cmd	:= DWORD_TO_BYTE(MesCmd_old[KK])	;
	
						END_IF	
						
						IF nSCO_Cmd.7 THEN
							; // code for select bit
						END_IF
						
						// create activation confirmation asdu
						stTxAsdu := stRxAsdu;
						stTxAsdu.info.stream.data[0] := nSCO_Cmd;	// Permet de mettre à jour que si pas en local
						stTxAsdu.ident.eCOT := eIEC870_COT_ACT_CON; //cause of transfer -> activation confirmation
						
						IF IN_Local THEN
							stTxAsdu.ident.bPN :=  TRUE;
						ELSE 
							stTxAsdu.ident.bPN := FALSE;
						END_IF						
						
						fbBuffer.TxAddObj(	putObj := stTxAsdu,
											buffer := stBuffer);
						IF NOT fbBuffer.bOk THEN
							// code for buffer overflow
							EXIT; 
						END_IF
						
						
						IF NOT nSCO_Cmd.7 AND NOT IN_Local THEN
							stTxAsdu := stRxAsdu;
							stTxAsdu.ident.eCOT := eIEC870_COT_ACT_TERM; // cause of transfer -> activation termination
							stTxAsdu.ident.bPN := FALSE;
							fbBuffer.TxAddObj(	putObj := stTxAsdu,
												buffer := stBuffer);
							IF NOT fbBuffer.bOk THEN
								// code for buffer overflow
								EXIT; 
							END_IF				
						END_IF
							
					END_IF
				END_FOR
				
